// TIA Portal V17 program export: 24 tag tables, 3 data types, 17 data blocks, 29 code blocks (in call order from the OBs), 32 instance data blocks

VAR_GLOBAL   // PLC tag table "Default tag table"
   OutputPin2 AT %QB147 : Byte;
   Tag_2 AT %QB152 : Byte;
   Tag_3 AT %QB155 : Byte;
   Tag_4 AT %QB154 : Byte;
   Tag_5 AT %QB153 : Byte;
   System_Byte AT %MB0 : Byte;
   DiagStatusUpdate AT %M0.1 : Bool;
   Tag_6 AT %MW122 : UInt;
END_VAR

VAR_GLOBAL   // PLC tag table "DCmotorControlMemory"
   motorBackwardMotion AT %M1551.2 : Bool;
   motorForwardMotion AT %M1550.7 : Bool;
   motorOpposite AT %M1551.4 : Bool;
   motorMovementActive AT %M1550.6 : Bool;
   hmiTestLeftMotorAlignment AT %M1551.6 : Bool;
   hmiTestRightTrackAlignment AT %M1551.7 : Bool;
   motorDirection AT %M1550.4 : Bool;
   highPulseDone AT %M1550.5 : Bool;
   reset AT %M1552.0 : Bool;
   direction1Pulse AT %MW1500 : Int;
   ctuReset1 AT %M1550.3 : Bool;
   motorPulseWidthSelector AT %M1551.5 : Bool;
   motorPulseWIidth AT %MD1534 : DInt;
   motorCycleTime AT %MD1530 : DInt;
   motorPulseQuantity AT %MW1502 : Int;
   activateMotorOperation AT %M1550.0 : Bool;
   hmiMoveMotorForward AT %M1552.1 : Bool;
   hmiMoveMotorBackward AT %M1552.2 : Bool;
   moveMotorForward AT %M1550.1 : Bool;
   moveMotorBackward AT %M1550.2 : Bool;
   leftTrackAlignmentComplete AT %M1551.1 : Bool;
   rightTrackAlignmentComplete AT %M1551.0 : Bool;
END_VAR

VAR_GLOBAL   // PLC tag table "EKSMemory"
   userIsLogged AT %M2150.0 : Bool;
   eksUserLevel AT %MB2101 : SInt;
   ActualAuthorizationLevel AT %MB2100 : SInt;
END_VAR

VAR_GLOBAL   // PLC tag table "HMIMemory"
   currentModel AT %MW3000 : Int;
   hmiButtonVisualization AT %M3050.6 : Bool;
   previousModel AT %MW3008 : Int;
   currentStep AT %MW3002 : Int;
   numberOfStepsToMove AT %MW3006 : UInt;
   stepToDivide AT %MW3012 : UInt;
   stepToInsert AT %MW3014 : UInt;
   hmiScreenNumber AT %MW3004 : Int;
   allowedTextChange AT %M3050.0 : Bool;
   progressBarMultiply AT %MW3010 : Int;
   lastCycleInputs AT %MD3034 : DInt;
   energySavingElapsedTime AT %MD3030 : Time;
   f7Button AT %M3050.5 : Bool;
   sequencerCopySequence AT %M3050.7 : Bool;
   codeReaderConfigurationVisible AT %M3050.2 : Bool;
   analogConfigurationVisible AT %M3050.1 : Bool;
   directAlarm AT %M3050.3 : Bool;
   directHome AT %M3050.4 : Bool;
   hmiRetractClampsReady AT %M3051.0 : Bool;
END_VAR

VAR_GLOBAL   // PLC tag table "alarmMemory"
   alarm0 AT %MW100 : Int;   // alarm number
   alarm1 AT %MW102 : Int;   // alarm number
   alarm2 AT %MW104 : Int;
   retIolink AT %MW108 : Int;
   retManifold AT %MW112 : Int;
   retEuchner AT %MW106 : Int;
   retIolink2 AT %MW110 : Int;
   QuitarErrorEscaner AT %MW6 : Word;
   bypass4 AT %M2.3 : Bool;
   bypass5 AT %M2.4 : Bool;
   retPrinter AT %MW114 : Int;
   reProfinetIO1 AT %MW116 : Int;
   reProfinetIO2 AT %MW118 : Int;
   reProfinetIO3 AT %MW120 : Int;
END_VAR

VAR_GLOBAL   // PLC tag table "analogAnalysisMemory"
   leftDistanceOk AT %M1700.4 : Bool;
   rightDistanceOk AT %M1700.5 : Bool;
   leftDistanceOk2 AT %M1700.7 : Bool;
   rightDistanceOk2 AT %M1701.0 : Bool;
   initialAlignmentOK AT %M1700.1 : Bool;
   initialPositionLeftTrackOK AT %M1700.2 : Bool;
   initialPositionRightTrackOK AT %M1700.3 : Bool;
   rightDistanceNormalizedValue AT %MD1660 : Real;
   leftDistanceNormalizedValue AT %MD1664 : Real;
   leftDistanceScaledValue AT %MD1668 : Real;
   rightDistanceScaledValue AT %MD1672 : Real;
   leftEffortOk AT %M1700.0 : Bool;
   rightEffortOk AT %M1700.6 : Bool;
   leftLoadCellSensorValue AT %MW1600 : Int;
   rightLoadCellSensorValue AT %MW1602 : Int;
   leftLoadCellNormalizedValue AT %MD1676 : Real;
   rightLoadCellNormalizedValue AT %MD1680 : Real;
   leftLoadCellScaledValue AT %MD1684 : Real;
   rightLoadCellScaledValue AT %MD1688 : Real;
   leftEffortNok AT %M1701.1 : Bool;
   rightEffortNok AT %M1701.2 : Bool;
   leftTrackRemoveMessage AT %M1701.3 : Bool;
   rightTrackRemoveMessage AT %M1701.4 : Bool;
   leftLoadCellHMIStatus AT %MW1604 : Int;
   rightLoadCellHMIStatus AT %MW1606 : Int;
   leftLoadCellHMIValue AT %MD1692 : Real;
   rightLoadCellHMIValue AT %MD1696 : Real;
END_VAR

VAR_GLOBAL   // PLC tag table "clockMemory"
   Clocks200ms_FP AT %M1.1 : Bool;
   Clocks400ms_FP AT %M1.2 : Bool;
   Clocks500ms_FP AT %M1.3 : Bool;
   Clocks800ms_FP AT %M1.4 : Bool;
   Clocks1s_FP AT %M1.5 : Bool;
   Clocks1600ms_FP AT %M1.6 : Bool;
   Clocks2s_FP AT %M1.7 : Bool;
   Clocks100ms_FP AT %M1.0 : Bool;
END_VAR

VAR_GLOBAL   // PLC tag table "codeReaderMemory"
   reqScannerConfig AT %M2250.2 : Bool;
   bufferReset AT %M2250.0 : Bool;
   idleTime AT %M2250.1 : Bool;
   rightTrackLabelIdentified AT %M2250.5 : Bool;
   leftTrackLabelIdentified AT %M2250.3 : Bool;
   motorLabelIdentified AT %M2250.4 : Bool;
   labelNOK AT %M2250.6 : Bool;
   labelOK AT %M2250.7 : Bool;
   trackLabelReadOutOfNest AT %M2251.0 : Bool;
   plasticBridgeLabelReadOutOfNest AT %M2251.1 : Bool;
END_VAR

VAR_GLOBAL   // PLC tag table "modeMemory"
   automaticMode AT %M3.0 : Bool;   // AUTO = 1
   manualMode AT %M3.1 : Bool;
   noMode AT %M3.2 : Bool;
   modelChangePermit AT %M187.1 : Bool;
END_VAR

VAR_GLOBAL   // PLC tag table "permissionMemory"
   maintenacePermission AT %M4.4 : Bool;
   adminPermission AT %M4.0 : Bool;
   lgPermission AT %M4.3 : Bool;
   gapLeaderPermission AT %M4.2 : Bool;
   editingPermission AT %M4.1 : Bool;
END_VAR

VAR_GLOBAL   // PLC tag table "printerMemory"
   reqPrint AT %M4000.0 : Bool;
   reqLastLabel AT %M4000.1 : Bool;
   resetPrinterErrors AT %M4000.2 : Bool;
   printBlackLabel AT %M4000.3 : Bool;
   resetPrinterCounter AT %M4000.4 : Bool;
   hmiSavePrinterReference AT %M4000.5 : Bool;
   hmiReadPrinterReference AT %M4000.6 : Bool;
END_VAR

VAR_GLOBAL   // PLC tag table "productionMemory"
   shift1Production AT %MW300 : Int;
   shift1 AT %M350.0 : Bool;
   shift2Production AT %MW302 : Int;
   shift2 AT %M350.1 : Bool;
   shift3Production AT %MW304 : Int;
   shift3 AT %M350.2 : Bool;
   timeShift1 AT %M350.3 : Bool;
   timeShift2 AT %M350.4 : Bool;
   timeShift3 AT %M350.5 : Bool;
END_VAR

VAR_GLOBAL   // PLC tag table "programMemory"
   cycleTimeReset AT %M250.1 : Bool;
   clearData AT %M250.0 : Bool;
   programAutoModeSelection AT %M250.3 : Bool;
   productInNest AT %M250.2 : Bool;
   bypass1 AT %M2.0 : Bool;
   bypass2 AT %M2.1 : Bool;
   bypass3 AT %M2.2 : Bool;
END_VAR

VAR_GLOBAL   // PLC tag table "pulses"
   hmiPulseInt AT %MD2000 : DInt;
   HMICycleCounterRestartPulse AT %M2004.4 : Bool;
   mode01SelectedPulse AT %M2004.6 : Bool;
   model02SelectedPulse AT %M2004.7 : Bool;
   model03SelectedPulse AT %M2005.0 : Bool;
   model04SelectedPulse AT %M2005.1 : Bool;
   model05SelectedPulse AT %M2005.2 : Bool;
   model06SelectedPulse AT %M2005.3 : Bool;
   model07SelectedPulse AT %M2005.4 : Bool;
   model08SelectedPulse AT %M2005.5 : Bool;
   model09SelectedPulse AT %M2005.6 : Bool;
   model10SelectedPulse AT %M2005.7 : Bool;
   model11SelectedPulse AT %M2006.0 : Bool;
   model12SelectedPulse AT %M2006.1 : Bool;
   model13SelectedPulse AT %M2006.2 : Bool;
   model14SelectedPulse AT %M2006.3 : Bool;
   model15SelectedPulse AT %M2006.4 : Bool;
   alarmPresentPulse AT %M2004.3 : Bool;
   "1stShiftChangePulse" AT %M2004.0 : Bool;
   "2ndShiftChangePulse" AT %M2004.1 : Bool;
   "3rdShiftChangePulse" AT %M2004.2 : Bool;
   stepChangeTimerResetInputPulse AT %M2009.4 : Bool;
   stepChangeTimerResetOutputPulse AT %M2009.5 : Bool;
   stationTurnedOffInSequencePulse AT %M2009.3 : Bool;
   model32SelectedPulse AT %M2008.5 : Bool;
   model31SelectedPulse AT %M2008.4 : Bool;
   model30SelectedPulse AT %M2008.3 : Bool;
   model29SelectedPulse AT %M2008.2 : Bool;
   model27SelectedPulse AT %M2008.0 : Bool;
   model28SelectedPulse AT %M2008.1 : Bool;
   model26SelectedPulse AT %M2007.7 : Bool;
   model25SelectedPulse AT %M2007.6 : Bool;
   model24SelectedPulse AT %M2007.5 : Bool;
   model23SelectedPulse AT %M2007.4 : Bool;
   model22SelectedPulse AT %M2007.3 : Bool;
   model21SelectedPulse AT %M2007.2 : Bool;
   model20SelectedPulse AT %M2007.1 : Bool;
   model19SelectedPulse AT %M2007.0 : Bool;
   model18SelectedPulse AT %M2006.7 : Bool;
   model17SelectedPulse AT %M2006.6 : Bool;
   model16SelectedPulse AT %M2006.5 : Bool;
   scanner3DataLogPulse AT %M2009.2 : Bool;
   scanner2DataLogPulse AT %M2009.1 : Bool;
   scanner1DataLogPulse AT %M2009.0 : Bool;
   motorScannerPulse AT %M2008.6 : Bool;
   rightTrackScannerPulse AT %M2008.7 : Bool;
   leftTrackScannerPulse AT %M2004.5 : Bool;
   scannerOk1Pulse AT %M2009.6 : Bool;
   scannerOk2Pulse AT %M2009.7 : Bool;
   scannerOk3Pulse AT %M2010.0 : Bool;
   leftTrackNokAlarmPulse AT %M2010.1 : Bool;
   rightTrackNokAlarmPulse AT %M2010.2 : Bool;
END_VAR

VAR_GLOBAL   // PLC tag table "sequenceMemory"
   aa AT %MW1104 : Int;
   a_correctas AT %MW1100 : Int;
   a_estados AT %MW1102 : Int;
   verificacion_estados_A AT %MW1114 : Int;
   verificacion_estados_B AT %MW1116 : Int;
   b_estados AT %MW1106 : Int;
   numberOfCorrectOutputStates AT %MW1110 : Int;
   bb AT %MW1108 : Int;
   previousStep AT %MW1112 : Int;
   sequenceRestart AT %M1150.0 : Bool;
   stationTurnedOffInSequence AT %M1150.1 : Bool;
END_VAR

VAR_GLOBAL   // PLC tag table "systemMemory"
   firstScan AT %M0.0 : Bool;
   LOG1 AT %M0.2 : Bool;
   LOG0 AT %M0.3 : Bool;
END_VAR

VAR_GLOBAL   // PLC tag table "EKSFieldbusInputs"
   iEKSLevel AT %IB201 : Byte;
   iEKSChipInside AT %I200.1 : Bool;
   iEKSEmployeeNumber AT %ID221 : DWord;
   iEKSKeyID1 AT %ID320 : DWord;
   iEKSKeyID2 AT %ID324 : DWord;
   iEKSJobFinished AT %I200.6 : Bool;
END_VAR

VAR_GLOBAL   // PLC tag table "safetyControllerFieldbusInputs"
   iSecurityEnabled AT %I46.0 : Bool;
   iEmergencyStop AT %I62.0 : Bool;
   iEmergencyStopMonitor AT %I62.1 : Bool;
   iOutputsEnabled AT %I82.0 : Bool;
END_VAR

VAR_GLOBAL   // PLC tag table "analogPLCInputs"
   iLeftLoadCell AT %IW13 : Int;
   iRightLoadCell AT %IW15 : Int;
   iRightDistanceSensor AT %IW17 : Int;
   iLeftDistanceSensor AT %IW19 : UInt;
END_VAR

VAR_GLOBAL   // PLC tag table "digitalFieldbusInputs"
   iRightTrackClampExt AT %I147.0 : Bool;
   iLeftTrackClampExt AT %I147.1 : Bool;
   iRightNestLocatingPinExt AT %I147.2 : Bool;
   iLeftNestLocatingPinExt AT %I147.3 : Bool;
   iRightTrackClampRet AT %I148.0 : Bool;
   iLeftTrackClampRet AT %I148.1 : Bool;
   iRightNestLocatingPinRet AT %I148.2 : Bool;
   iLeftNestLocatingPinRet AT %I148.3 : Bool;
   iLeftTrackPS1 AT %I149.0 : Bool;
   iLeftTrackPS2 AT %I149.1 : Bool;
   iRightTrackPS1 AT %I149.2 : Bool;
   iRightTrackPS2 AT %I149.3 : Bool;
   iLeftNestInitialPos AT %I149.4 : Bool;
   iRightNestInitialPos AT %I149.5 : Bool;
   iRightManualClampClosed AT %I149.6 : Bool;
   iLeftManualClampClosed AT %I149.7 : Bool;
   iPlasticBridgePS AT %I151.0 : Bool;
   iLeftNestWorkingPos AT %I151.1 : Bool;
   iPokayokeLeftTrackPS AT %I151.2 : Bool;
   iPokayokeRightTrackPS AT %I151.3 : Bool;
   iPlasticBridgeClampClosed AT %I151.4 : Bool;
   iInsertPlasticBridgePos AT %I151.6 : Bool;
   iInsertShaftPos AT %I151.7 : Bool;
END_VAR

VAR_GLOBAL   // PLC tag table "digitalPLCInputs"
   iAirPreassureSensor AT %I0.1 : Bool;
   iMotorConnected AT %I0.2 : Bool;
   iRestartButton AT %I0.0 : Bool;
   iMotorRelayStatus AT %I0.3 : Bool;
END_VAR

VAR_GLOBAL   // PLC tag table "digitalFielbusOutputs"
   qCylinder1DirectionA AT %Q149.0 : Bool;
   qCylinder1DirectionB AT %Q151.0 : Bool;
   qCylinder2DirectionA AT %Q149.1 : Bool;
   qCylinder2DirectionB AT %Q151.1 : Bool;
   qCylinder7DirectionA AT %Q149.6 : Bool;
   qCylinder7DirectionB AT %Q151.6 : Bool;
   qCylinder4DirectionA AT %Q149.3 : Bool;
   qCylinder4DirectionB AT %Q151.3 : Bool;
   qCylinder5DirectionA AT %Q149.4 : Bool;
   qCylinder5DirectionB AT %Q151.4 : Bool;
   qCylinder6DirectionA AT %Q149.5 : Bool;
   qCylinder6DirectionB AT %Q151.5 : Bool;
   qCylinder3DirectionA AT %Q149.2 : Bool;
   qCylinder3DirectionB AT %Q151.2 : Bool;
   qCylinder8DirectionA AT %Q149.7 : Bool;
   qCylinder8DirectionB AT %Q151.7 : Bool;
   qCylinder9DirectionA AT %Q148.0 : Bool;
   qCylinder9DirectionB AT %Q150.0 : Bool;
   qCylinder10DirectionA AT %Q148.1 : Bool;
   qCylinder10DirectionB AT %Q150.1 : Bool;
   qActivateCutOffValve AT %Q147.0 : Bool;
END_VAR

VAR_GLOBAL   // PLC tag table "digitalPLCOutputs"
   qAirInletValve AT %Q0.0 : Bool;
   qLampActivation AT %Q0.4 : Bool;
   qFanActivation AT %Q0.5 : Bool;
   qRedStacklight AT %Q1.7 : Bool;
   qYellowStacklight AT %Q1.6 : Bool;
   qGreenStacklight AT %Q1.5 : Bool;
   qControlIN AT %Q0.6 : Bool;
   qActiveMotor AT %Q0.7 : Bool;
   qDirectionChange AT %Q1.0 : Bool;
   qRedIndicator AT %Q1.1 : Bool;
   qGreenIndicator AT %Q1.2 : Bool;
   qYellowIndicator AT %Q1.3 : Bool;
   qBlueStacklight AT %Q1.4 : Bool;
END_VAR

VAR_GLOBAL   // PLC tag table "EKSFieldbusOutputs"
   qEKSStartAddress AT %QB201 : Byte;
   qEKSDataLength AT %QB202 : Byte;
   qEKSData1 AT %QB204 : Byte;
   qEKSData2 AT %QB205 : Byte;
   qEKSWriteCMD AT %Q200.0 : Bool;
END_VAR

TYPE "udtButtons"
// stored: IsFailsafeCompliant false
   STRUCT
      bReq : Bool;
      bP : Bool;
      bTGG : Bool;
      bCmd : Bool;
      bAkn : Bool;
      b1 : Bool;
      b2 : Bool;
      b3 : Bool;
   END_STRUCT;
END_TYPE

TYPE "udt_EKS_KEY"
// stored: IsFailsafeCompliant false
   STRUCT
      ID1 : DWord;   // Key unique ID [bytes 1-4]
      ID2 : DWord;   // Key unique ID [bytes 5-8]
      EMPLOYEE_ID : DWord;   // Employee ID number [hex format]
      LEVEL : Int;   // Key level stored inside key
      COMMENTS : WString[10];   // Comments of the key
      _res_1 : Int;
   END_STRUCT;
END_TYPE

TYPE "udt_referenceMainInfo"
// stored: IsFailsafeCompliant false
   STRUCT
      id : Int;
      description : String[20];
      partNumber : String[8];
      rev : String[2];
      customerNumber : String[8];
      vpps : String[14];
      locationCode : String[1];
      dataIdentifier : String[3];
      duns : String[9];
   END_STRUCT;
END_TYPE

DATA_BLOCK "DB_REC_IJCORE"   // DB1006
{ S7_Optimized_Access := 'FALSE' }
VERSION : 0.1
// stored: AutoNumber false, DBAccessibleFromOPCUA true, DBAccessibleFromWebserver true, IsOnlyStoredInLoadMemory false, IsWriteProtectedInAS false
   VAR
      SW_Message : Array[1..300] of Word;
      Message : Array[1..50] of Struct
         Answer : Int;
         Content : Array[1..30] of Byte;
      END_STRUCT;
   END_VAR
BEGIN
   SW_Message[1..8] := 16#FFFF;
   SW_Message[9..300] := 16#0000;
   Message[1..50].Answer := 0;
   Message[1].Content[1..30] := 16#00;
   Message[2].Content[1..30] := 16#00;
   Message[3].Content[1..30] := 16#00;
   Message[4].Content[1..30] := 16#00;
   Message[5].Content[1..30] := 16#00;
   Message[6].Content[1..30] := 16#00;
   Message[7].Content[1..30] := 16#00;
   Message[8].Content[1..30] := 16#00;
   Message[9].Content[1..30] := 16#00;
   Message[10].Content[1..30] := 16#00;
   Message[11].Content[1..30] := 16#00;
   Message[12].Content[1..30] := 16#00;
   Message[13].Content[1..30] := 16#00;
   Message[14].Content[1..30] := 16#00;
   Message[15].Content[1..30] := 16#00;
   Message[16].Content[1..30] := 16#00;
   Message[17].Content[1..30] := 16#00;
   Message[18].Content[1..30] := 16#00;
   Message[19].Content[1..30] := 16#00;
   Message[20].Content[1..30] := 16#00;
   Message[21].Content[1..30] := 16#00;
   Message[22].Content[1..30] := 16#00;
   Message[23].Content[1..30] := 16#00;
   Message[24].Content[1..30] := 16#00;
   Message[25].Content[1..30] := 16#00;
   Message[26].Content[1..30] := 16#00;
   Message[27].Content[1..30] := 16#00;
   Message[28].Content[1..30] := 16#00;
   Message[29].Content[1..30] := 16#00;
   Message[30].Content[1..30] := 16#00;
   Message[31].Content[1..30] := 16#00;
   Message[32].Content[1..30] := 16#00;
   Message[33].Content[1..30] := 16#00;
   Message[34].Content[1..30] := 16#00;
   Message[35].Content[1..30] := 16#00;
   Message[36].Content[1..30] := 16#00;
   Message[37].Content[1..30] := 16#00;
   Message[38].Content[1..30] := 16#00;
   Message[39].Content[1..30] := 16#00;
   Message[40].Content[1..30] := 16#00;
   Message[41].Content[1..30] := 16#00;
   Message[42].Content[1..30] := 16#00;
   Message[43].Content[1..30] := 16#00;
   Message[44].Content[1..30] := 16#00;
   Message[45].Content[1..30] := 16#00;
   Message[46].Content[1..30] := 16#00;
   Message[47].Content[1..30] := 16#00;
   Message[48].Content[1..30] := 16#00;
   Message[49].Content[1..30] := 16#00;
   Message[50].Content[1..30] := 16#00;
END_DATA_BLOCK

DATA_BLOCK "DB_SEND_IJCORE"   // DB1005
{ S7_Optimized_Access := 'FALSE' }
VERSION : 0.1
// stored: AutoNumber false, DBAccessibleFromOPCUA true, DBAccessibleFromWebserver true, IsOnlyStoredInLoadMemory false, IsWriteProtectedInAS false
   VAR
      Awake_DW : Word := 16#0000;
      Awake_SW : Int := 1;
      SW_Message : Array[1..300] of Word;
      Message : Array[1..50] of Struct
         Content : Array[1..80] of Byte;
      END_STRUCT;
   END_VAR
BEGIN
   SW_Message[1..8] := 16#FFFF;
   SW_Message[9..300] := 16#0000;
   Message[1].Content[1..80] := 16#00;
   Message[2].Content[1..80] := 16#00;
   Message[3].Content[1..80] := 16#00;
   Message[4].Content[1..80] := 16#00;
   Message[5].Content[1..80] := 16#00;
   Message[6].Content[1..80] := 16#00;
   Message[7].Content[1..80] := 16#00;
   Message[8].Content[1..80] := 16#00;
   Message[9].Content[1..80] := 16#00;
   Message[10].Content[1..80] := 16#00;
   Message[11].Content[1..80] := 16#00;
   Message[12].Content[1..80] := 16#00;
   Message[13].Content[1..80] := 16#00;
   Message[14].Content[1..80] := 16#00;
   Message[15].Content[1..80] := 16#00;
   Message[16].Content[1..80] := 16#00;
   Message[17].Content[1..80] := 16#00;
   Message[18].Content[1..80] := 16#00;
   Message[19].Content[1..80] := 16#00;
   Message[20].Content[1..80] := 16#00;
   Message[21].Content[1..80] := 16#00;
   Message[22].Content[1..80] := 16#00;
   Message[23].Content[1..80] := 16#00;
   Message[24].Content[1..80] := 16#00;
   Message[25].Content[1..80] := 16#00;
   Message[26].Content[1..80] := 16#00;
   Message[27].Content[1..80] := 16#00;
   Message[28].Content[1..80] := 16#00;
   Message[29].Content[1..80] := 16#00;
   Message[30].Content[1..80] := 16#00;
   Message[31].Content[1..80] := 16#00;
   Message[32].Content[1..80] := 16#00;
   Message[33].Content[1..80] := 16#00;
   Message[34].Content[1..80] := 16#00;
   Message[35].Content[1..80] := 16#00;
   Message[36].Content[1..80] := 16#00;
   Message[37].Content[1..80] := 16#00;
   Message[38].Content[1..80] := 16#00;
   Message[39].Content[1..80] := 16#00;
   Message[40].Content[1..80] := 16#00;
   Message[41].Content[1..80] := 16#00;
   Message[42].Content[1..80] := 16#00;
   Message[43].Content[1..80] := 16#00;
   Message[44].Content[1..80] := 16#00;
   Message[45].Content[1..80] := 16#00;
   Message[46].Content[1..80] := 16#00;
   Message[47].Content[1..80] := 16#00;
   Message[48].Content[1..80] := 16#00;
   Message[49].Content[1..80] := 16#00;
   Message[50].Content[1..80] := 16#00;
END_DATA_BLOCK

DATA_BLOCK "model"   // DB5
{ S7_Optimized_Access := 'TRUE' }
VERSION : 0.1
// stored: AutoNumber false, DBAccessibleFromOPCUA true, DBAccessibleFromWebserver true, IsOnlyStoredInLoadMemory false, IsRetainMemResEnabled false, IsWriteProtectedInAS false, MemoryReserve 100
   VAR RETAIN
      "name" : Array[0..32] of String[50];
   END_VAR
   VAR
      day : Int := 2;
      dayText : String := '    11';
      month : Int := 8;
      monthText : String := '     8';
      year : Int := 2012;
      yearReady : String := '2012';
      hour : Int := 17;
      hourText : String := '    17';
      minutes : Int := 30;
      minutesText : String := '    30';
      seconds : Int := 30;
      secondsText : String := '    31';
      active : Array[0..32] of Bool;
   END_VAR
   VAR RETAIN
      datum1 : Array[0..32] of String[50];
      datum2 : Array[0..32] of String[50];
      datum3 : Array[0..32] of String[50];
      datum4 : Array[0..32] of String[50];
      datum5 : Array[0..32] of String[50];
      datum6 : Array[0..32] of String[50];
      datum7 : Array[0..32] of String[50];
      Description : Array[0..32] of String[50];
   END_VAR
BEGIN
   "name"[0..1] := '4118099';
   "name"[2] := '4118098';
   "name"[3..32] := '';
   active[0] := FALSE;
   active[1..2] := TRUE;
   active[3..32] := FALSE;
   datum1[0..2] := 'Z';
   datum1[3] := 'ddd';
   datum1[4..17] := 'Z';
   datum1[18..32] := '';
   datum2[0..17] := '410';
   datum2[18..32] := '';
   datum3[0..17] := '6';
   datum3[18..32] := '';
   datum4[0..2] := 'BACKREST W33A POWER MEMO L6';
   datum4[3] := 'prueba';
   datum4[4] := 'outter trackw33';
   datum4[5..16] := 'BACKREST W33A POWER MEMO L6';
   datum4[17] := 'P42LHNOMEM';
   datum4[18..32] := '';
   datum5[0] := '2389161X-01';
   datum5[1..2] := '2521784';
   datum5[3] := '2389161X-01';
   datum5[4..5] := '2282685X-01';
   datum5[6..16] := '2521784';
   datum5[17] := '2418723X-01';
   datum5[18..32] := '';
   datum6[0..32] := '';
   datum7[0..32] := '';
   Description[0..1] := 'H-Frame 4W RH';
   Description[2] := 'H-Frame 4W LH';
   Description[3..32] := '';
END_DATA_BLOCK

DATA_BLOCK "retentiveValues"   // DB54
{ S7_Optimized_Access := 'TRUE' }
VERSION : 0.1
// stored: AutoNumber true, DBAccessibleFromOPCUA true, DBAccessibleFromWebserver true, IsOnlyStoredInLoadMemory false, IsRetainMemResEnabled true, IsWriteProtectedInAS false, MemoryReserve 100, RetainMemoryReserve 0
   VAR RETAIN
      stationInSequence : Bool := FALSE;
   END_VAR
BEGIN
END_DATA_BLOCK

DATA_BLOCK "analog"   // DB3
{ S7_Optimized_Access := 'TRUE' }
VERSION : 0.1
// stored: AutoNumber false, DBAccessibleFromOPCUA true, DBAccessibleFromWebserver true, IsOnlyStoredInLoadMemory false, IsRetainMemResEnabled false, IsWriteProtectedInAS false, MemoryReserve 100
   VAR RETAIN
      value1 : Array[0..32] of Real;   // Setpoint del valor analógico 1 [modelo]
      low1 : Array[0..32] of Real;   // Valor bajo del valor analógico 1 [modelo]
      high1 : Array[0..32] of Real;   // Valor alto del valor analógico 1 [modelo]
      value2 : Array[0..32] of Real;
      low2 : Array[0..32] of Real;
      high2 : Array[0..32] of Real;
      value3 : Array[0..32] of Real;
      low3 : Array[0..32] of Real;
      high3 : Array[0..32] of Real;
      value4 : Array[0..32] of Real;
      low4 : Array[0..32] of Real;
      high4 : Array[0..32] of Real;
      value5 : Array[0..32] of Real;
      low5 : Array[0..32] of Real;
      high5 : Array[0..32] of Real;
      value6 : Array[0..32] of Real;
      low6 : Array[0..32] of Real;
      high6 : Array[0..32] of Real;
      value7 : Array[0..32] of Real;
      low7 : Array[0..32] of Real;
      high7 : Array[0..32] of Real;
      value8 : Array[0..32] of Real;
      low8 : Array[0..32] of Real;
      high8 : Array[0..32] of Real;
      value9 : Array[0..32] of Real;
      low9 : Array[0..32] of Real;
      high9 : Array[0..32] of Real;
      value10 : Array[0..32] of Real;
      low10 : Array[0..32] of Real;
      high10 : Array[0..32] of Real;
      text : Array[0..10] of String;
      analog1 : Bool := TRUE;
      analog2 : Bool := TRUE;
      analog3 : Bool := TRUE;
      analog4 : Bool := TRUE;
      analog5 : Bool := FALSE;
      analog6 : Bool := FALSE;
   END_VAR
   VAR
      visibility : Array[0..6] of Bool;
      current1 : Int := 0;
      current2 : Int := 0;
      current3 : Int := 0;
      current4 : Int := 0;
      current5 : Int := 0;
      current6 : Int := 0;
      laserConstant : Real := 0.005802801;
      okDistance : Bool := FALSE;
      nest1 : Array[0..5] of Int;
      nest2 : Array[0..5] of Int;
      nest3 : Array[0..5] of Int;
      nest4 : Array[0..5] of Int;
      motorCounter : Int := 1600;
   END_VAR
   VAR RETAIN
      motorQuantity : Int := 0;
   END_VAR
   VAR
      analogReading1 : Array[0..9] of Real;
      analogReading2 : Array[0..9] of Real;
      leftLoadCellMaxValueObtained : Real := 0.0;
      rightLoadCellMaxValueObtained : Real := 0.0;
   END_VAR
BEGIN
   value1[0..3] := -63.9458;
   value1[4] := -16.86112;
   value1[5..8] := -63.9458;
   value1[9..14] := 131.4746;
   value1[15] := 340.0;
   value1[16] := -17.19834;
   value1[17..19] := 131.4746;
   value1[20..32] := 0.0;
   low1[0..2] := -1.0;
   low1[3] := 120.0;
   low1[4] := 154.0;
   low1[5] := 100.0;
   low1[6..8] := 72.0;
   low1[9..13] := 120.0;
   low1[14] := 153.0;
   low1[15] := 0.0;
   low1[16..17] := 120.0;
   low1[18] := 154.0;
   low1[19] := 120.0;
   low1[20..32] := 0.0;
   high1[0..2] := 2.0;
   high1[3] := 5.0;
   high1[4] := 2.0;
   high1[5] := 110.0;
   high1[6..8] := 76.0;
   high1[9..13] := 5.0;
   high1[14] := 2.0;
   high1[15] := 41.1;
   high1[16..17] := 5.0;
   high1[18] := 2.0;
   high1[19] := 5.0;
   high1[20..32] := 0.0;
   value2[0..3] := -65.29469;
   value2[4] := -17.51449;
   value2[5..8] := -65.29469;
   value2[9..14] := 131.4746;
   value2[15] := 340.0;
   value2[16] := -17.40911;
   value2[17..19] := 131.4746;
   value2[20..32] := 0.0;
   low2[0..2] := -1.0;
   low2[3] := 60.0;
   low2[4] := 154.0;
   low2[5] := 100.0;
   low2[6..8] := 60.0;
   low2[9..13] := 0.0;
   low2[14] := 153.0;
   low2[15..17] := 0.0;
   low2[18] := 154.0;
   low2[19..32] := 0.0;
   high2[0..2] := 2.0;
   high2[3] := 75.0;
   high2[4] := 2.0;
   high2[5] := 110.0;
   high2[6..8] := 64.0;
   high2[9..13] := 5.0;
   high2[14] := 2.0;
   high2[15] := 38.7;
   high2[16..17] := 5.0;
   high2[18] := 2.0;
   high2[19] := 5.0;
   high2[20..32] := 0.0;
   value3[0..3] := 16#0000_02E7;
   value3[4] := 16#0000_01DE;
   value3[5..8] := 16#0000_02E7;
   value3[9..14] := 16#0000_01DE;
   value3[15..16] := 16#0000_DDDE;
   value3[17..19] := 16#0000_01DE;
   value3[20..32] := 0.0;
   low3[0..2] := 200.0;
   low3[3] := 40.0;
   low3[4] := 0.0;
   low3[5] := 200.0;
   low3[6..8] := 40.0;
   low3[9..32] := 0.0;
   high3[0..2] := 500.0;
   high3[3] := 250.0;
   high3[4] := 0.0;
   high3[5] := 210.0;
   high3[6..8] := 250.0;
   high3[9..32] := 0.0;
   value4[0..19] := 40.0;
   value4[20..32] := 0.0;
   low4[0..2] := 200.0;
   low4[3] := 40.0;
   low4[4] := 0.0;
   low4[5] := 200.0;
   low4[6..8] := 40.0;
   low4[9..32] := 0.0;
   high4[0..2] := 500.0;
   high4[3] := 250.0;
   high4[4] := 3.0;
   high4[5] := 210.0;
   high4[6..8] := 250.0;
   high4[9..19] := 3.0;
   high4[20..32] := 0.0;
   value5[0..14] := 3.0;
   value5[15] := 8.0;
   value5[16..19] := 3.0;
   value5[20..32] := 0.0;
   low5[0..32] := 0.0;
   high5[0..19] := 59.0;
   high5[20..32] := 0.0;
   value6[0..32] := 0.0;
   low6[0..32] := 0.0;
   high6[0..32] := 0.0;
   value7[0..3] := -65.29469;
   value7[4] := -16.90327;
   value7[5..8] := -65.29469;
   value7[9..14] := -16.86112;
   value7[15] := 0.0;
   value7[16] := -17.19834;
   value7[17..19] := -16.86112;
   value7[20..32] := 0.0;
   low7[0..3] := 142.0;
   low7[4] := 125.0;
   low7[5..8] := 142.0;
   low7[9..13] := 0.0;
   low7[14] := 26.0;
   low7[15..17] := 0.0;
   low7[18] := 128.0;
   low7[19..32] := 0.0;
   high7[0..3] := 2.0;
   high7[4] := 3.0;
   high7[5..13] := 2.0;
   high7[14] := 5.0;
   high7[15] := 0.0;
   high7[16..19] := 2.0;
   high7[20..32] := 0.0;
   value8[0..3] := -65.29469;
   value8[4] := -17.17727;
   value8[5..8] := -65.29469;
   value8[9..14] := -17.17727;
   value8[15] := 0.0;
   value8[16] := -17.51449;
   value8[17..19] := -17.17727;
   value8[20..32] := 0.0;
   low8[0..3] := 142.0;
   low8[4] := 125.0;
   low8[5..8] := 142.0;
   low8[9..13] := 0.0;
   low8[14] := 26.0;
   low8[15..17] := 0.0;
   low8[18] := 128.0;
   low8[19..32] := 0.0;
   high8[0..3] := 2.0;
   high8[4] := 3.0;
   high8[5..13] := 2.0;
   high8[14] := 5.0;
   high8[15] := 0.0;
   high8[16..19] := 2.0;
   high8[20..32] := 0.0;
   value9[0..3] := 1.348892;
   value9[4] := 0.6533699;
   value9[5..8] := 1.348892;
   value9[9..32] := 0.0;
   low9[0..32] := 0.0;
   high9[0..3] := 0.0;
   high9[4] := 2.0;
   high9[5..13] := 0.0;
   high9[14] := 2.0;
   high9[15..17] := 0.0;
   high9[18] := 2.0;
   high9[19..32] := 0.0;
   value10[0..3] := 0.0;
   value10[4] := 0.2739925;
   value10[5..8] := 0.0;
   value10[9..14] := 0.3161469;
   value10[15..16] := 0.0;
   value10[17..19] := 0.3161469;
   value10[20..32] := 0.0;
   low10[0..32] := 0.0;
   high10[0..17] := 0.0;
   high10[18] := 2.0;
   high10[19..32] := 0.0;
   text[0] := '';
   text[1] := 'Distancia Izquierda';
   text[2] := 'Distancia Derecha';
   text[3] := 'Esfuerzo Izquierdo';
   text[4] := 'Esfuerzo Derecho';
   text[5..6] := '';
   text[7] := 'Final izquierdo';
   text[8] := 'Final derecho';
   text[9] := 'Alineacion inicial';
   text[10] := 'Alineacion final';
   visibility[0] := FALSE;
   visibility[1..4] := TRUE;
   visibility[5..6] := FALSE;
   nest1[0..5] := 0;
   nest2[0..5] := 0;
   nest3[0..5] := 0;
   nest4[0..5] := 0;
   analogReading1[0..2] := 58.96373;
   analogReading1[3] := 0.4987493;
   analogReading1[4] := 0.0;
   analogReading1[5..9] := 58.96373;
   analogReading2[0..9] := 0.0;
END_DATA_BLOCK

DATA_BLOCK "eks"   // DB305
{ S7_Optimized_Access := 'FALSE' }
VERSION : 0.1
// stored: AutoNumber false, DBAccessibleFromOPCUA true, DBAccessibleFromWebserver true, IsOnlyStoredInLoadMemory false, IsWriteProtectedInAS false
   VAR RETAIN
      status : Struct
         operator : Bool := TRUE;
         gapLeader : Bool := TRUE;
         maintenance : Bool := TRUE;
         administrator : Bool := TRUE;
         spare4 : Bool := FALSE;
         spare5 : Bool := FALSE;
         spare6 : Bool := FALSE;
         spare7 : Bool := FALSE;
         addModeEnabled : Bool := TRUE;
         addMode : Bool := FALSE;
         reset : Bool := FALSE;
         nbMaxAchieved : Bool := FALSE;
         fpStoreKeyIn : Bool := FALSE;
         spare15 : Bool := FALSE;
         spare16 : Bool := FALSE;
         spare17 : Bool := FALSE;
      END_STRUCT;
      hmi : Struct
         operatorKey : Bool := FALSE;
         addMode : Bool := FALSE;
         endAddMode : Bool := FALSE;
         writeKeyNewLevel : Bool := FALSE;
         writeKewKeyID : Bool := FALSE;
         updateNbAdmin : Bool := FALSE;
         spare6 : Bool := FALSE;
         spare7 : Bool := FALSE;
         spare10 : Bool := FALSE;
         spare11 : Bool := FALSE;
         spare12 : Bool := FALSE;
         spare13 : Bool := FALSE;
         spare14 : Bool := FALSE;
         spare15 : Bool := FALSE;
         spare16 : Bool := FALSE;
         spare17 : Bool := FALSE;
      END_STRUCT;
      timeout : Struct
         resetSet : Int := 9999;
         resetStatus : Int := 9100;
      END_STRUCT;
      pageIndex : Int := 1;   // Index of the page of HMI
      saveLine : Int := 0;   // Line to save key
      removeLine : Int := 0;   // Line to remove key
      actualLevel : Int := 5;   // Actual level of key
      nbAdmin : Int := 30740;   // Number of admin counted
      tCycle : Int := 0;   // Index for function Cycle (look for key)
      nbMaxAdmin : Int := 5;   // Number of administrator max
      savedPageNumber : Word := 16#0001;
      sparesBlock1 : Array[22..47] of Byte;   // Reserve
      insertedKey { S7_SetPoint := 'True'} : "udt_EKS_KEY";   // Information of Key Inserted
      hmiPage { S7_SetPoint := 'True'} : Array[1..10] of "udt_EKS_KEY";   // Information displayed on HMI
      spareBlock2 : Array[270..299] of Byte;   // Reserve
      keys { S7_SetPoint := 'True'} : Array[1..130] of "udt_EKS_KEY";
      deleteKeys : "udt_EKS_KEY";
   END_VAR
BEGIN
   sparesBlock1[22..47] := 16#00;
   insertedKey.ID1 := 16#6B8F_0010;
   insertedKey.ID2 := 16#3200_0000;
   insertedKey.EMPLOYEE_ID := 16#0000_0000;
   insertedKey.LEVEL := 5;
   insertedKey.COMMENTS := WSTRING#'ADMIN';
   insertedKey._res_1 := 0;
   hmiPage[1].ID1 := 16#27A0_0010;
   hmiPage[2].ID1 := 16#8DDD_0010;
   hmiPage[3].ID1 := 16#9750_0010;
   hmiPage[4].ID1 := 16#4D33_0010;
   hmiPage[5].ID1 := 16#7650_0010;
   hmiPage[6].ID1 := 16#6B8F_0010;
   hmiPage[7].ID1 := 16#3A6D_0010;
   hmiPage[8..10].ID1 := 16#0000_0000;
   hmiPage[1..7].ID2 := 16#3200_0000;
   hmiPage[8..10].ID2 := 16#0000_0000;
   hmiPage[1].EMPLOYEE_ID := 16#0001_0000;
   hmiPage[2].EMPLOYEE_ID := 16#0000_0001;
   hmiPage[3].EMPLOYEE_ID := 16#0000_0002;
   hmiPage[4..5].EMPLOYEE_ID := 16#0000_0000;
   hmiPage[6].EMPLOYEE_ID := 16#0000_0200;
   hmiPage[7].EMPLOYEE_ID := 16#0000_0100;
   hmiPage[8..10].EMPLOYEE_ID := 16#0000_0000;
   hmiPage[1].LEVEL := 5;
   hmiPage[2].LEVEL := 2;
   hmiPage[3].LEVEL := 3;
   hmiPage[4].LEVEL := 5;
   hmiPage[5].LEVEL := 3;
   hmiPage[6].LEVEL := 5;
   hmiPage[7].LEVEL := 3;
   hmiPage[8..10].LEVEL := 0;
   hmiPage[1].COMMENTS := WSTRING#'CESAR';
   hmiPage[2].COMMENTS := WSTRING#'GAP';
   hmiPage[3].COMMENTS := WSTRING#'MANT';
   hmiPage[4..5].COMMENTS := WSTRING#'CESAR';
   hmiPage[6].COMMENTS := WSTRING#'ADMIN';
   hmiPage[7].COMMENTS := WSTRING#'MANT';
   hmiPage[8..10].COMMENTS := WSTRING#'';
   hmiPage[1..10]._res_1 := 0;
   spareBlock2[270..299] := 16#00;
   keys[1].ID1 := 16#27A0_0010;
   keys[2].ID1 := 16#8DDD_0010;
   keys[3].ID1 := 16#9750_0010;
   keys[4].ID1 := 16#4D33_0010;
   keys[5].ID1 := 16#7650_0010;
   keys[6].ID1 := 16#6B8F_0010;
   keys[7].ID1 := 16#3A6D_0010;
   keys[8..109].ID1 := 16#0000_0000;
   keys[110].ID1 := 16#DB52_0010;
   keys[111..130].ID1 := 16#0000_0000;
   keys[1..7].ID2 := 16#3200_0000;
   keys[8..109].ID2 := 16#0000_0000;
   keys[110].ID2 := 16#3200_0000;
   keys[111..130].ID2 := 16#0000_0000;
   keys[1].EMPLOYEE_ID := 16#0001_0000;
   keys[2].EMPLOYEE_ID := 16#0000_0001;
   keys[3].EMPLOYEE_ID := 16#0000_0002;
   keys[4..5].EMPLOYEE_ID := 16#0000_0000;
   keys[6].EMPLOYEE_ID := 16#0000_0200;
   keys[7].EMPLOYEE_ID := 16#0000_0100;
   keys[8..130].EMPLOYEE_ID := 16#0000_0000;
   keys[1].LEVEL := 5;
   keys[2].LEVEL := 2;
   keys[3].LEVEL := 3;
   keys[4].LEVEL := 5;
   keys[5].LEVEL := 3;
   keys[6].LEVEL := 5;
   keys[7].LEVEL := 3;
   keys[8..109].LEVEL := 0;
   keys[110].LEVEL := 5;
   keys[111..130].LEVEL := 0;
   keys[1].COMMENTS := WSTRING#'CESAR';
   keys[2].COMMENTS := WSTRING#'GAP';
   keys[3].COMMENTS := WSTRING#'MANT';
   keys[4..5].COMMENTS := WSTRING#'CESAR';
   keys[6].COMMENTS := WSTRING#'ADMIN';
   keys[7].COMMENTS := WSTRING#'MANT';
   keys[8..109].COMMENTS := WSTRING#'';
   keys[110].COMMENTS := WSTRING#'Robins';
   keys[111..130].COMMENTS := WSTRING#'';
   keys[1..130]._res_1 := 0;
   deleteKeys.ID1 := 16#0000_0000;
   deleteKeys.ID2 := 16#0000_0000;
   deleteKeys.EMPLOYEE_ID := 16#0000_0000;
   deleteKeys.LEVEL := 0;
   deleteKeys.COMMENTS := WSTRING#'';
   deleteKeys._res_1 := 0;
END_DATA_BLOCK

DATA_BLOCK "motor"   // DB19
{ S7_Optimized_Access := 'TRUE' }
VERSION : 0.1
// stored: AutoNumber true, DBAccessibleFromOPCUA true, DBAccessibleFromWebserver true, IsOnlyStoredInLoadMemory false, IsRetainMemResEnabled false, IsWriteProtectedInAS false, MemoryReserve 100
   VAR RETAIN
      on : Bool := TRUE;
      track1Test : Bool := FALSE;
      track2Test : Bool := FALSE;
      pulseNumber1 : Int := 5;
      waitTime1 : DInt := 100;
      pulseWidth2 : DInt := 10;
      cicleTime2 : DInt := 200;
      pulseNumber2 : Int := 5;
      waitTime2 : DInt := 100;
      cicleTime1 : DInt := 200;
      pulseWidth1 : DInt := 10;
   END_VAR
BEGIN
END_DATA_BLOCK

DATA_BLOCK "step"   // DB4
{ S7_Optimized_Access := 'TRUE' }
VERSION : 0.1
// stored: AutoNumber false, DBAccessibleFromOPCUA true, DBAccessibleFromWebserver true, IsOnlyStoredInLoadMemory false, IsRetainMemResEnabled false, IsWriteProtectedInAS false, MemoryReserve 100
   VAR RETAIN
      "time" : Array[0..32, 0..25] of Int;   // Tiempo de duración de cada paso [modelo, paso]
      number : Array[0..32] of Int;   // Número de pasos por modelo
   END_VAR
   VAR
      stepChangeTimer : DInt := 0;
      stepChangeTimerStart : Bool := FALSE;
      counterDone : Bool := FALSE;
   END_VAR
BEGIN
   "time"[0,0] := 0;
   "time"[0,1..5] := 500;
   "time"[0,6] := 1000;
   "time"[0,7] := 500;
   "time"[0,8] := 1000;
   "time"[0,9..10] := 500;
   "time"[0,11..25] := 0;
   "time"[1,0] := 0;
   "time"[1,1..5] := 500;
   "time"[1,6] := 1000;
   "time"[1,7] := 500;
   "time"[1,8] := 1000;
   "time"[1,9..10] := 500;
   "time"[1,11..25] := 0;
   "time"[2,0] := 0;
   "time"[2,1..5] := 500;
   "time"[2,6] := 1000;
   "time"[2,7] := 500;
   "time"[2,8] := 1000;
   "time"[2,9..10] := 500;
   "time"[2,11..25] := 0;
   "time"[3,0] := 0;
   "time"[3,1] := 500;
   "time"[3,2..4] := 1500;
   "time"[3,5..11] := 500;
   "time"[3,12..25] := 0;
   "time"[4,0] := 0;
   "time"[4,1] := 500;
   "time"[4,2..4] := 1500;
   "time"[4,5..11] := 500;
   "time"[4,12..25] := 0;
   "time"[5,0] := 0;
   "time"[5,1] := 1000;
   "time"[5,2] := 0;
   "time"[5,3] := 1000;
   "time"[5,4..25] := 0;
   "time"[6,0] := 0;
   "time"[6,1..2] := 1500;
   "time"[6,3] := 0;
   "time"[6,4..9] := 3000;
   "time"[6,10..25] := 0;
   "time"[7,0] := 0;
   "time"[7,1..2] := 1500;
   "time"[7,3] := 0;
   "time"[7,4..9] := 3000;
   "time"[7,10..25] := 0;
   "time"[8,0] := 0;
   "time"[8,1..2] := 1500;
   "time"[8,3] := 0;
   "time"[8,4..9] := 3000;
   "time"[8,10..25] := 0;
   "time"[9,0..3] := 0;
   "time"[9,4..5] := 500;
   "time"[9,6..25] := 0;
   "time"[10,0..3] := 0;
   "time"[10,4..5] := 500;
   "time"[10,6..25] := 0;
   "time"[11,0..3] := 0;
   "time"[11,4..5] := 500;
   "time"[11,6..25] := 0;
   "time"[12,0..3] := 0;
   "time"[12,4..5] := 500;
   "time"[12,6..25] := 0;
   "time"[13,0..3] := 0;
   "time"[13,4..5] := 500;
   "time"[13,6..25] := 0;
   "time"[14,0..3] := 0;
   "time"[14,4..5] := 500;
   "time"[14,6..25] := 0;
   "time"[15,0..25] := 0;
   "time"[16,0..3] := 0;
   "time"[16,4..5] := 500;
   "time"[16,6..25] := 0;
   "time"[17,0..3] := 0;
   "time"[17,4..5] := 500;
   "time"[17,6..25] := 0;
   "time"[18,0..3] := 0;
   "time"[18,4..5] := 500;
   "time"[18,6..25] := 0;
   "time"[19,0..3] := 0;
   "time"[19,4..5] := 500;
   "time"[19,6..25] := 0;
   "time"[20,0..25] := 0;
   "time"[21,0..25] := 0;
   "time"[22,0..25] := 0;
   "time"[23,0..25] := 0;
   "time"[24,0..25] := 0;
   "time"[25,0..25] := 0;
   "time"[26,0..25] := 0;
   "time"[27,0..25] := 0;
   "time"[28,0..25] := 0;
   "time"[29,0..25] := 0;
   "time"[30,0..25] := 0;
   "time"[31,0..25] := 0;
   "time"[32,0..25] := 0;
   number[0..2] := 10;
   number[3..4] := 11;
   number[5] := 3;
   number[6..14] := 9;
   number[15] := 8;
   number[16..19] := 9;
   number[20..32] := 0;
END_DATA_BLOCK

DATA_BLOCK "labels"   // DB6
{ S7_Optimized_Access := 'TRUE' }
VERSION : 0.1
// stored: AutoNumber false, DBAccessibleFromOPCUA true, DBAccessibleFromWebserver true, IsOnlyStoredInLoadMemory false, IsRetainMemResEnabled false, IsWriteProtectedInAS false, MemoryReserve 100
   VAR RETAIN
      label1 : Array[0..32] of String[50];   // Etiqueta 1
      label2 : Array[0..32] of String[50];
      label3 : Array[0..32] of String[50];
      label4 : Array[0..32] of String[50];
      label5 : Array[0..32] of String[50];
      label6 : Array[0..32] of String[50];
      posLabel1 : Array[0..32] of Int;   // Posición de etiqueta 1
      posLabel2 : Array[0..32] of Int;
      posLabel3 : Array[0..32] of Int;
      posLabel4 : Array[0..32] of Int;
      posLabel5 : Array[0..32] of Int;
      posLabel6 : Array[0..32] of Int;
      text : Array[0..5] of String;   // Texto HMI de etiquetas
   END_VAR
   VAR
      done2 : Bool := FALSE;
      errorPort2 : Bool := FALSE;
      statusPort2 : Word := 16#7000;
      statusReset : Word := 16#7000;
   END_VAR
   VAR RETAIN
      doneReset : Bool := FALSE;
      scanner1 : Bool := TRUE;
      scanner2 : Bool := TRUE;
      scanner3 : Bool := TRUE;
      scanner4 : Bool := FALSE;
      scanner5 : Bool := FALSE;
   END_VAR
   VAR
      scanner6 : Bool := FALSE;
      scannerOn : Bool := TRUE;
      codeScanned : String := ' ';
      codeReceived : String := '';
      ndr : Bool := FALSE;
      error : Bool := FALSE;
      status : Word := 16#7002;
      lenght : UInt := 0;
      lablelBlock : Array[0..6] of Bool;
      nestScannerRead : String := ' ';
      readScanner : String := '03804073GO23548$R';
      extraction : Array[0..6] of String;
      previousBarcode : String := '';
   END_VAR
BEGIN
   label1[0..4] := '038';
   label1[5] := '1';
   label1[6..8] := '038';
   label1[9] := '202';
   label1[10..11] := '592';
   label1[12] := '202';
   label1[13] := '592';
   label1[14] := '202';
   label1[15..16] := '';
   label1[17] := '592';
   label1[18] := '202';
   label1[19] := '592';
   label1[20..32] := '';
   label2[0..1] := '4066654';
   label2[2] := '4066308';
   label2[3] := '4066654';
   label2[4] := '4066308';
   label2[5] := '2';
   label2[6..7] := '709';
   label2[8] := '706';
   label2[9] := '723';
   label2[10] := '724';
   label2[11] := '723';
   label2[12] := '724';
   label2[13] := '769';
   label2[14] := '768';
   label2[15..16] := '';
   label2[17..18] := '685';
   label2[19] := '163';
   label2[20..32] := '';
   label3[0..1] := '4066430';
   label3[2] := '4066646';
   label3[3] := '4066430';
   label3[4] := '4066646';
   label3[5] := '3';
   label3[6..7] := '708';
   label3[8] := '707';
   label3[9] := '718';
   label3[10] := '719';
   label3[11] := '718';
   label3[12..14] := '719';
   label3[15..16] := '';
   label3[17..18] := '680';
   label3[19] := '161';
   label3[20..32] := '';
   label4[0..32] := '';
   label5[0..32] := '';
   label6[0..32] := '';
   posLabel1[0..14] := 1;
   posLabel1[15..16] := 0;
   posLabel1[17..19] := 1;
   posLabel1[20..32] := 0;
   posLabel2[0..4] := 1;
   posLabel2[5] := 2;
   posLabel2[6..8] := 10;
   posLabel2[9..12] := 5;
   posLabel2[13..14] := 1;
   posLabel2[15..16] := 0;
   posLabel2[17..19] := 5;
   posLabel2[20..32] := 0;
   posLabel3[0..4] := 1;
   posLabel3[5] := 3;
   posLabel3[6..8] := 10;
   posLabel3[9..13] := 5;
   posLabel3[14] := 13;
   posLabel3[15..16] := 0;
   posLabel3[17..19] := 5;
   posLabel3[20..32] := 0;
   posLabel4[0..32] := 0;
   posLabel5[0..32] := 0;
   posLabel6[0..32] := 0;
   text[0] := '';
   text[1] := 'Motor';
   text[2] := 'Track Izq';
   text[3] := 'Track der';
   text[4..5] := '';
   lablelBlock[0] := FALSE;
   lablelBlock[1..3] := TRUE;
   lablelBlock[4..6] := FALSE;
   extraction[0] := '';
   extraction[1] := '038';
   extraction[2..3] := '0380407';
   extraction[4..6] := '';
END_DATA_BLOCK

DATA_BLOCK "conveyor"   // DB41
{ S7_Optimized_Access := 'FALSE' }
VERSION : 0.1
// stored: AutoNumber true, DBAccessibleFromOPCUA true, DBAccessibleFromWebserver true, IsOnlyStoredInLoadMemory false, IsWriteProtectedInAS false
   VAR
      printLabel : Bool := FALSE;
      description : String := 'BACKREST W33A POWER MEMO L6';
      partNumber : String := '2389161X-01';
      lastScann : String := '03804073GO23548$R';
      okModelBit : Bool := FALSE;
      leftTrackScan : String := '4066654X016PN4O385$R';
      rightTrackScan : String := '4066430X016LN4S161$R';
      motorScan : String := '03804073GO23548$R';
   END_VAR
BEGIN
END_DATA_BLOCK

DATA_BLOCK "dataLogging"   // DB36
{ S7_Optimized_Access := 'TRUE' }
VERSION : 0.1
// stored: AutoNumber true, DBAccessibleFromOPCUA true, DBAccessibleFromWebserver true, IsOnlyStoredInLoadMemory false, IsRetainMemResEnabled false, IsWriteProtectedInAS false, MemoryReserve 100
   VAR
      scanning : Array[1..3] of String;
      alignment : Real := 0.0;
      pieceOk : Bool := FALSE;
   END_VAR
BEGIN
   scanning[1] := '03804073GO23548$R';
   scanning[2] := '4066654X016PN4O385$R';
   scanning[3] := '4066430X016LN4S161$R';
END_DATA_BLOCK

DATA_BLOCK "DB_PrinterReference"   // DB33
{ S7_Optimized_Access := 'TRUE' }
VERSION : 0.1
// stored: AutoNumber true, DBAccessibleFromOPCUA true, DBAccessibleFromWebserver true, IsOnlyStoredInLoadMemory false, IsRetainMemResEnabled false, IsWriteProtectedInAS false, MemoryReserve 100
   VAR
      reference : Array[0..32] of "udt_referenceMainInfo";
   END_VAR
BEGIN
   reference[0..32].id := 0;
   reference[0..32].description := '';
   reference[0..32].partNumber := '';
   reference[0..32].rev := '';
   reference[0..32].customerNumber := '';
   reference[0..32].vpps := '';
   reference[0..32].locationCode := '';
   reference[0..32].dataIdentifier := '';
   reference[0..32].duns := '';
END_DATA_BLOCK

DATA_BLOCK "devicesAlarm"   // DB37
{ S7_Optimized_Access := 'TRUE' }
VERSION : 0.1
// stored: AutoNumber true, DBAccessibleFromOPCUA true, DBAccessibleFromWebserver true, IsOnlyStoredInLoadMemory false, IsRetainMemResEnabled false, IsWriteProtectedInAS false, MemoryReserve 100
   VAR
      bannerStatus : Array[0..1023] of Bool;
      manifold : Array[0..1023] of Bool;
      iolink1 : Array[0..1023] of Bool;
      profinetIO1 : Array[0..1023] of Bool;
      profinetIO2 : Array[0..1023] of Bool;
      profinetIO3 : Array[0..1023] of Bool;
      printer : Array[0..1023] of Bool;
      printerDiag : DIS;
   END_VAR
BEGIN
   bannerStatus[0..1023] := FALSE;
   manifold[0..1023] := FALSE;
   iolink1[0..1023] := FALSE;
   profinetIO1[0..1023] := FALSE;
   profinetIO2[0..1023] := FALSE;
   profinetIO3[0..1023] := FALSE;
   printer[0..1023] := FALSE;
   printerDiag.MaintainanceState := 16#0000_0000;
   printerDiag.ComponentStateDetail := 16#0000_8000;
   printerDiag.OwnState := 0;
   printerDiag.IOState := 16#0001;
   printerDiag.OperatingState := 0;
END_DATA_BLOCK

DATA_BLOCK "hmi"   // DB7
{ S7_Optimized_Access := 'TRUE' }
VERSION : 0.1
// stored: AutoNumber true, DBAccessibleFromOPCUA true, DBAccessibleFromWebserver true, IsOnlyStoredInLoadMemory false, IsRetainMemResEnabled false, IsWriteProtectedInAS false, MemoryReserve 100
   VAR
      modeButton : Bool := FALSE;
      mode : Int := 2;
      model : Array[0..32] of Bool;
      recipeStep : Int := 9;
      "a" : DInt := 44690590;
      "b" : DInt := 536_871_082;
      mascA : DInt := 66846862;
      mascB : DInt := 0;
      recipeStepTime : Int := 500;
      recipeStepSubstract : Bool := FALSE;
      recipeStepAdd : Bool := FALSE;
      recipeLastStep : Int := 9;
      updateStep : Bool := FALSE;
      moveToCurrentStep : Bool := FALSE;
      recordA1 : Bool := FALSE;
      readA1 : Bool := FALSE;
      recordA2 : Bool := FALSE;
      readA2 : Bool := FALSE;
      recordB1 : Bool := FALSE;
      readB1 : Bool := FALSE;
      recordB2 : Bool := FALSE;
      readB2 : Bool := FALSE;
      recordAnalog : Bool := FALSE;
      readAnalog : Bool := FALSE;
      recipeStepQuantity : Int := 10;
      eraseStep : Bool := FALSE;
      insertStep : Bool := FALSE;
      copyStep : Bool := FALSE;
      copySequence : Bool := FALSE;
      copySequenceStep : Bool := FALSE;
      baseStep : Int := 10;
      destinationStep : Int := 11;
      baseModel : Int := 7;
      destinationModel : Int := 8;
      baseModelStep : Int := 0;
      modelDestinationStep : Int := 0;
      baseModelStep_1 : Int := 2;
      modelDestinationStep_1 : Int := 3;
      operatorTextIndicator : String := ' ';
      enableStationAir : Bool := FALSE;
      enableAirHmiPermission : Bool := FALSE;
      insertAlarmKey : Bool := FALSE;
      enableStationVisualizationButton : Bool := FALSE;
      enableStationHideAlarmButton : Bool := FALSE;
      alarmAckmowledge : Bool := FALSE;
      home : Bool := FALSE;
      advancePercentage : Real := 0.0;
      administratorAlarmButton : Bool := FALSE;
      activateLamp : Bool := FALSE;
      activateFan : Bool := TRUE;
   END_VAR
   VAR RETAIN
      cicles : Int := 444;
      production1 : Int := 80;
      production2 : Int := 48;
      production3 : Int := 17;
   END_VAR
   VAR
      productionRestart1 : Bool := FALSE;
      productionRestart2 : Bool := FALSE;
      productionRestart3 : Bool := FALSE;
      cyclesRestart : Bool := FALSE;
      manualPrint : Bool := FALSE;
      BLOQUEO : Bool := TRUE;
      manualModeNecessary : Bool := FALSE;
      modelChange : Bool := FALSE;
      alarmManualButton : Bool := FALSE;
      user : String := 'Administrator';
      pass : String := 'PASSWORD';
   END_VAR
BEGIN
   model[0..32] := FALSE;
END_DATA_BLOCK

DATA_BLOCK "sensorDistribution"   // DB129
{ S7_Optimized_Access := 'TRUE' }
VERSION : 0.1
// stored: AutoNumber false, DBAccessibleFromOPCUA true, DBAccessibleFromWebserver true, IsOnlyStoredInLoadMemory false, IsRetainMemResEnabled false, IsWriteProtectedInAS false, MemoryReserve 100
   VAR
      inputsStatus : Array[0..31] of Byte;
      outputsStatus : Array[0..31] of Byte;
   END_VAR
BEGIN
   inputsStatus[0..5] := 16#00;
   inputsStatus[6] := 16#01;
   inputsStatus[7] := 16#00;
   inputsStatus[8] := 16#01;
   inputsStatus[9..16] := 16#00;
   inputsStatus[17..18] := 16#01;
   inputsStatus[19..31] := 16#00;
   outputsStatus[0] := 16#01;
   outputsStatus[1] := 16#00;
   outputsStatus[2] := 16#01;
   outputsStatus[3] := 16#00;
   outputsStatus[4] := 16#01;
   outputsStatus[5] := 16#00;
   outputsStatus[6] := 16#01;
   outputsStatus[7..31] := 16#00;
END_DATA_BLOCK

DATA_BLOCK "inputs"   // DB1
{ S7_Optimized_Access := 'TRUE' }
VERSION : 0.1
// stored: AutoNumber false, DBAccessibleFromOPCUA true, DBAccessibleFromWebserver true, IsOnlyStoredInLoadMemory false, IsRetainMemResEnabled false, IsWriteProtectedInAS false, MemoryReserve 100
   VAR RETAIN
      inputSequence : Array[0..32, 0..25] of DInt;   // 32 entradas [modelo, paso]
   END_VAR
   VAR
      activeInputsReq : Array[0..31] of Bool;
   END_VAR
   VAR RETAIN
      maskSequence : Array[0..32, 0..25] of DInt;   // Máscara de entradas
   END_VAR
   VAR
      activeMask : Array[0..31] of Bool;
   END_VAR
   VAR RETAIN
      inputText : Array[0..31] of String;   // Texto HMI de cada entrada
   END_VAR
   VAR
      buttonStatus : Array[0..63] of Bool;
      activeInputsReqDInt : DInt := 131392;   // Estado de sensores en directo
      inputActive : Array[0..31] of Bool;
      euchnerReading : Array[0..254] of Char;
      nestScannerReading : String := '';
      upperScannerReading : String := '';
      nestScanerReceived : Array[0..254] of Char;
      nestScanerReceivedString : String := '';
      upperScannerReceived : Array[0..254] of Char;
      upperScannerReceivedString : String := '';
      euchnerReadingString : String := '$01';
      laserReading : Word := 16#0000;
      laserConstant : Real := 0.0005802801;
      laserReadingInt : DInt := 0;
      readingConversion : LReal := 0.0;
      euchnerName : String := '';
      euchner : Array[0..257] of Byte;
   END_VAR
BEGIN
   inputSequence[0,0] := 23724353;
   inputSequence[0,1] := 827_518_278;
   inputSequence[0,2..4] := 44756294;
   inputSequence[0,5] := 1_252_650_334;
   inputSequence[0,6..7] := 1_118_432_670;
   inputSequence[0,8] := 1_118_432_414;
   inputSequence[0,9] := 44690590;
   inputSequence[0,10] := 44892160;
   inputSequence[0,11..25] := 0;
   inputSequence[1,0] := 23724353;
   inputSequence[1,1] := 827_518_278;
   inputSequence[1,2..4] := 44756294;
   inputSequence[1,5] := 1_252_650_334;
   inputSequence[1,6..7] := 1_118_432_670;
   inputSequence[1,8] := 1_118_432_414;
   inputSequence[1,9] := 44690590;
   inputSequence[1,10] := 44892160;
   inputSequence[1,11..25] := 0;
   inputSequence[2,0] := 23724353;
   inputSequence[2,1] := 827_514_182;
   inputSequence[2,2..4] := 44752198;
   inputSequence[2,5] := 1_252_646_238;
   inputSequence[2,6..7] := 1_118_428_574;
   inputSequence[2,8] := 1_118_428_318;
   inputSequence[2,9] := 44686494;
   inputSequence[2,10] := 44892160;
   inputSequence[2,11..25] := 0;
   inputSequence[3,0] := 23724353;
   inputSequence[3,1] := 827_518_278;
   inputSequence[3,2..4] := 44756294;
   inputSequence[3,5] := 1_252_650_334;
   inputSequence[3,6..8] := 1_118_432_670;
   inputSequence[3,9] := 1_118_432_414;
   inputSequence[3,10] := 44690590;
   inputSequence[3,11] := 44892160;
   inputSequence[3,12..25] := 0;
   inputSequence[4,0] := 23724353;
   inputSequence[4,1] := 827_514_182;
   inputSequence[4,2..4] := 44752198;
   inputSequence[4,5] := 1_252_646_238;
   inputSequence[4,6..7] := 1_118_428_574;
   inputSequence[4,8] := 1_118_428_446;
   inputSequence[4,9] := 1_118_428_318;
   inputSequence[4,10] := 44686494;
   inputSequence[4,11] := 44892160;
   inputSequence[4,12..25] := 0;
   inputSequence[5,0..1] := 64;
   inputSequence[5,2..3] := 128;
   inputSequence[5,4..25] := 0;
   inputSequence[6,0] := 23724353;
   inputSequence[6,1] := 827_780_422;
   inputSequence[6,2] := 44756294;
   inputSequence[6,3] := 44755974;
   inputSequence[6,4] := 1_252_650_334;
   inputSequence[6,5..7] := 1_118_432_670;
   inputSequence[6,8] := 1_118_432_414;
   inputSequence[6,9] := 44630336;
   inputSequence[6,10..25] := 0;
   inputSequence[7,0] := 23724353;
   inputSequence[7,1] := 827_780_422;
   inputSequence[7,2] := 44756294;
   inputSequence[7,3] := 44755974;
   inputSequence[7,4] := 1_252_650_334;
   inputSequence[7,5..7] := 1_118_432_670;
   inputSequence[7,8] := 1_118_432_414;
   inputSequence[7,9] := 44630336;
   inputSequence[7,10..25] := 0;
   inputSequence[8,0] := 23724353;
   inputSequence[8,1] := 827_776_326;
   inputSequence[8,2] := 44752198;
   inputSequence[8,3] := 44751878;
   inputSequence[8,4] := 1_252_646_238;
   inputSequence[8,5] := 1_118_428_574;
   inputSequence[8,6] := 1_118_428_318;
   inputSequence[8,7] := 1_118_428_574;
   inputSequence[8,8] := 1_118_428_318;
   inputSequence[8,9] := 44630336;
   inputSequence[8,10..25] := 0;
   inputSequence[9,0] := 321;
   inputSequence[9,1] := 4193656;
   inputSequence[9,2] := 2_017_459_576;
   inputSequence[9,3] := 1_077_935_482;
   inputSequence[9,4] := 1_073_745_282;
   inputSequence[9,5..6] := 1_073_745_538;
   inputSequence[9,7..9] := 320;
   inputSequence[9,10..25] := 0;
   inputSequence[10,0] := 321;
   inputSequence[10,1] := 4193656;
   inputSequence[10,2] := 2_017_459_576;
   inputSequence[10,3] := 1_077_935_482;
   inputSequence[10,4] := 1_073_745_282;
   inputSequence[10,5..6] := 1_073_745_538;
   inputSequence[10,7..9] := 320;
   inputSequence[10,10..25] := 0;
   inputSequence[11,0] := 321;
   inputSequence[11,1] := 4193656;
   inputSequence[11,2] := 2_017_459_576;
   inputSequence[11,3] := 1_077_935_482;
   inputSequence[11,4] := 1_073_745_282;
   inputSequence[11,5..6] := 1_073_745_538;
   inputSequence[11,7..9] := 320;
   inputSequence[11,10..25] := 0;
   inputSequence[12,0] := 321;
   inputSequence[12,1] := 8387960;
   inputSequence[12,2] := 2_021_653_880;
   inputSequence[12,3] := 1_082_129_786;
   inputSequence[12,4] := 1_077_939_586;
   inputSequence[12,5] := 1_077_939_842;
   inputSequence[12,6] := 1_073_745_538;
   inputSequence[12,7..9] := 320;
   inputSequence[12,10..25] := 0;
   inputSequence[13,0] := 321;
   inputSequence[13,1] := 4193656;
   inputSequence[13,2] := 2_017_459_576;
   inputSequence[13,3] := 1_077_935_482;
   inputSequence[13,4] := 1_073_745_282;
   inputSequence[13,5..6] := 1_073_745_538;
   inputSequence[13,7..9] := 320;
   inputSequence[13,10..25] := 0;
   inputSequence[14,0] := 321;
   inputSequence[14,1] := 4193656;
   inputSequence[14,2] := 2_017_459_576;
   inputSequence[14,3] := 1_077_935_482;
   inputSequence[14,4] := 1_073_745_282;
   inputSequence[14,5..6] := 1_073_745_538;
   inputSequence[14,7..9] := 320;
   inputSequence[14,10..25] := 0;
   inputSequence[15,0] := 11;
   inputSequence[15,1] := 63040522;
   inputSequence[15,2] := 1_338_108_938;
   inputSequence[15,3] := 65137674;
   inputSequence[15,4] := 65135628;
   inputSequence[15,5] := 65134612;
   inputSequence[15,6] := 57344;
   inputSequence[15,7] := 805_363_712;
   inputSequence[15,8] := 10;
   inputSequence[15,9..25] := 0;
   inputSequence[16,0] := 321;
   inputSequence[16,1] := 8387960;
   inputSequence[16,2] := 2_021_653_880;
   inputSequence[16,3] := 1_082_129_786;
   inputSequence[16,4] := 1_077_939_586;
   inputSequence[16,5] := 1_077_939_842;
   inputSequence[16,6] := 1_073_745_538;
   inputSequence[16,7..9] := 320;
   inputSequence[16,10..25] := 0;
   inputSequence[17,0] := 321;
   inputSequence[17,1] := 4193656;
   inputSequence[17,2] := 2_017_459_576;
   inputSequence[17,3] := 1_077_935_482;
   inputSequence[17,4] := 1_073_745_282;
   inputSequence[17,5..6] := 1_073_745_538;
   inputSequence[17,7..9] := 320;
   inputSequence[17,10..25] := 0;
   inputSequence[18,0] := 321;
   inputSequence[18,1] := 4193656;
   inputSequence[18,2] := 2_017_459_576;
   inputSequence[18,3] := 1_077_935_482;
   inputSequence[18,4] := 1_073_745_282;
   inputSequence[18,5..6] := 1_073_745_538;
   inputSequence[18,7..9] := 320;
   inputSequence[18,10..25] := 0;
   inputSequence[19,0] := 321;
   inputSequence[19,1] := 4193656;
   inputSequence[19,2] := 2_017_459_576;
   inputSequence[19,3] := 1_077_935_482;
   inputSequence[19,4] := 1_073_745_282;
   inputSequence[19,5..6] := 1_073_745_538;
   inputSequence[19,7..9] := 320;
   inputSequence[19,10..25] := 0;
   inputSequence[20,0..25] := 0;
   inputSequence[21,0..25] := 0;
   inputSequence[22,0..25] := 0;
   inputSequence[23,0..25] := 0;
   inputSequence[24,0..25] := 0;
   inputSequence[25,0..25] := 0;
   inputSequence[26,0..25] := 0;
   inputSequence[27,0..25] := 0;
   inputSequence[28,0..25] := 0;
   inputSequence[29,0..25] := 0;
   inputSequence[30,0..25] := 0;
   inputSequence[31,0..25] := 0;
   inputSequence[32,0..25] := 0;
   activeInputsReq[0] := TRUE;
   activeInputsReq[1..5] := FALSE;
   activeInputsReq[6] := TRUE;
   activeInputsReq[7] := FALSE;
   activeInputsReq[8] := TRUE;
   activeInputsReq[9..16] := FALSE;
   activeInputsReq[17] := TRUE;
   activeInputsReq[18] := FALSE;
   activeInputsReq[19] := TRUE;
   activeInputsReq[20] := FALSE;
   activeInputsReq[21..22] := TRUE;
   activeInputsReq[23] := FALSE;
   activeInputsReq[24] := TRUE;
   activeInputsReq[25..31] := FALSE;
   maskSequence[0,0] := 66859008;
   maskSequence[0,1] := 66846720;
   maskSequence[0,2] := 66847168;
   maskSequence[0,3..4] := 66846848;
   maskSequence[0,5..8] := 66846720;
   maskSequence[0,9] := 66846862;
   maskSequence[0,10] := 66649232;
   maskSequence[0,11..25] := 0;
   maskSequence[1,0] := 66859008;
   maskSequence[1,1] := 66846720;
   maskSequence[1,2] := 66847168;
   maskSequence[1,3..4] := 66846848;
   maskSequence[1,5..8] := 66846720;
   maskSequence[1,9] := 66846862;
   maskSequence[1,10] := 66649232;
   maskSequence[1,11..25] := 0;
   maskSequence[2,0] := 66859008;
   maskSequence[2,1] := 66846720;
   maskSequence[2,2] := 66847168;
   maskSequence[2,3..4] := 66846848;
   maskSequence[2,5..8] := 66846720;
   maskSequence[2,9] := 66846862;
   maskSequence[2,10] := 66649232;
   maskSequence[2,11..25] := 0;
   maskSequence[3,0] := 66859008;
   maskSequence[3,1] := 66846720;
   maskSequence[3,2] := 66847168;
   maskSequence[3,3..4] := 66846848;
   maskSequence[3,5..7] := 66846720;
   maskSequence[3,8] := 66846976;
   maskSequence[3,9] := 66846720;
   maskSequence[3,10] := 66846848;
   maskSequence[3,11] := 66649232;
   maskSequence[3,12..25] := 0;
   maskSequence[4,0] := 66859008;
   maskSequence[4,1] := 66846720;
   maskSequence[4,2] := 66847168;
   maskSequence[4,3..4] := 66846848;
   maskSequence[4,5..7] := 66846720;
   maskSequence[4,8] := 66847168;
   maskSequence[4,9] := 66846720;
   maskSequence[4,10] := 66846848;
   maskSequence[4,11] := 66649232;
   maskSequence[4,12..25] := 0;
   maskSequence[5,0..1] := -65;
   maskSequence[5,2..3] := -129;
   maskSequence[5,4..25] := 0;
   maskSequence[6,0..2] := 66846720;
   maskSequence[6,3] := 66847168;
   maskSequence[6,4..8] := 66846720;
   maskSequence[6,9] := 66847168;
   maskSequence[6,10..25] := 0;
   maskSequence[7,0..1] := 66846720;
   maskSequence[7,2..3] := 66847168;
   maskSequence[7,4..6] := 66846720;
   maskSequence[7,7] := 66846976;
   maskSequence[7,8] := 66846720;
   maskSequence[7,9] := 66847168;
   maskSequence[7,10..25] := 0;
   maskSequence[8,0..1] := 66846720;
   maskSequence[8,2..3] := 66847168;
   maskSequence[8,4..5] := 66846720;
   maskSequence[8,6..7] := 66846976;
   maskSequence[8,8] := 66846720;
   maskSequence[8,9] := 66847168;
   maskSequence[8,10..25] := 0;
   maskSequence[9,0] := -322;
   maskSequence[9,1] := 2_014_248_960;
   maskSequence[9,2..3] := 983040;
   maskSequence[9,4..5] := 79687736;
   maskSequence[9,6] := 134_213_948;
   maskSequence[9,7..8] := -2;
   maskSequence[9,9] := 134_217_406;
   maskSequence[9,10..25] := 0;
   maskSequence[10,0] := -322;
   maskSequence[10,1] := 2_014_289_920;
   maskSequence[10,2..3] := 1024000;
   maskSequence[10,4..5] := 79687736;
   maskSequence[10,6] := 134_213_948;
   maskSequence[10,7..8] := -2;
   maskSequence[10,9] := 134_217_406;
   maskSequence[10,10..25] := 0;
   maskSequence[11,0] := -322;
   maskSequence[11,1] := 2_014_248_960;
   maskSequence[11,2..3] := 983040;
   maskSequence[11,4..5] := 79687736;
   maskSequence[11,6] := 134_213_948;
   maskSequence[11,7..8] := -2;
   maskSequence[11,9] := 134_217_406;
   maskSequence[11,10..25] := 0;
   maskSequence[12,0] := -322;
   maskSequence[12,1] := 2_014_248_960;
   maskSequence[12,2..3] := 983040;
   maskSequence[12,4..5] := 79687736;
   maskSequence[12,6] := 134_213_948;
   maskSequence[12,7..8] := -2;
   maskSequence[12,9] := 134_217_406;
   maskSequence[12,10..25] := 0;
   maskSequence[13,0] := -322;
   maskSequence[13,1] := 2_014_248_960;
   maskSequence[13,2..3] := 983040;
   maskSequence[13,4..5] := 79687736;
   maskSequence[13,6] := 134_213_948;
   maskSequence[13,7..8] := -2;
   maskSequence[13,9] := 134_217_406;
   maskSequence[13,10..25] := 0;
   maskSequence[14,0] := -322;
   maskSequence[14,1] := 2_014_248_960;
   maskSequence[14,2] := 806_289_408;
   maskSequence[14,3] := 983040;
   maskSequence[14,4..5] := 79687736;
   maskSequence[14,6] := 134_213_948;
   maskSequence[14,7..8] := -2;
   maskSequence[14,9] := 134_217_406;
   maskSequence[14,10..25] := 0;
   maskSequence[15,0] := 0;
   maskSequence[15,1] := 2_080_374_784;
   maskSequence[15,2..3] := 805_306_368;
   maskSequence[15,4..5] := 868_220_928;
   maskSequence[15,6..7] := 268_435_452;
   maskSequence[15,8..25] := 0;
   maskSequence[16,0] := -322;
   maskSequence[16,1] := 2_014_248_960;
   maskSequence[16,2..3] := 983040;
   maskSequence[16,4..5] := 79687736;
   maskSequence[16,6] := 134_213_948;
   maskSequence[16,7..8] := -2;
   maskSequence[16,9] := 134_217_406;
   maskSequence[16,10..25] := 0;
   maskSequence[17,0] := -322;
   maskSequence[17,1] := 2_014_248_960;
   maskSequence[17,2..3] := 983040;
   maskSequence[17,4..5] := 79687736;
   maskSequence[17,6] := 134_213_948;
   maskSequence[17,7..8] := -2;
   maskSequence[17,9] := 134_217_406;
   maskSequence[17,10..25] := 0;
   maskSequence[18,0] := -322;
   maskSequence[18,1] := 2_014_248_960;
   maskSequence[18,2..3] := 983040;
   maskSequence[18,4..5] := 79687736;
   maskSequence[18,6] := 134_213_948;
   maskSequence[18,7..8] := -2;
   maskSequence[18,9] := 134_217_406;
   maskSequence[18,10..25] := 0;
   maskSequence[19,0] := -322;
   maskSequence[19,1] := 2_014_248_960;
   maskSequence[19,2..3] := 983040;
   maskSequence[19,4..5] := 79687736;
   maskSequence[19,6] := 134_213_948;
   maskSequence[19,7..8] := -2;
   maskSequence[19,9] := 134_217_406;
   maskSequence[19,10..25] := 0;
   maskSequence[20,0..25] := 0;
   maskSequence[21,0..25] := 0;
   maskSequence[22,0..25] := 0;
   maskSequence[23,0..25] := 0;
   maskSequence[24,0..25] := 0;
   maskSequence[25,0..25] := 0;
   maskSequence[26,0..25] := 0;
   maskSequence[27,0..25] := 0;
   maskSequence[28,0..25] := 0;
   maskSequence[29,0..25] := 0;
   maskSequence[30,0..25] := 0;
   maskSequence[31,0..25] := 0;
   maskSequence[32,0..25] := 0;
   activeMask[0..11] := FALSE;
   activeMask[12..13] := TRUE;
   activeMask[14..17] := FALSE;
   activeMask[18..25] := TRUE;
   activeMask[26..31] := FALSE;
   inputText[0] := 'CLEAR DATA';
   inputText[1] := 'Clamp izq. cerrado PRX18151';
   inputText[2] := 'Clamp der. cerrado PRX18150';
   inputText[3] := 'Clamp plastic bridge cerrado PRX19130';
   inputText[4] := 'Plastic bridge presente PRX19090';
   inputText[5] := 'Reserva';
   inputText[6] := 'Herramental izq. pos. inicio PRX18130';
   inputText[7] := 'Herramental izq pos trabajo PRX19091';
   inputText[8] := 'Herramental der. pos. inicio PRX18131';
   inputText[9] := 'Reserva';
   inputText[10] := 'Track 1 izq. presente PRX18090';
   inputText[11] := 'Track 1 der. presente PRX18110';
   inputText[12] := 'Tornillo track izq. PRX19110';
   inputText[13] := 'Tornillo track der. PRX19111';
   inputText[14] := 'Track 2 izq. presente PRX18091';
   inputText[15] := 'Track 2 der. presente PRX18111';
   inputText[16] := 'Posicion nido colocar track PRX19150';
   inputText[17] := 'Posicion nido ensamble varilla PRX19151';
   inputText[18] := 'Quitar pieza';
   inputText[19..26] := 'Reserva';
   inputText[27] := 'Escaner motor OK';
   inputText[28] := 'Escaner Track izq OK';
   inputText[29] := 'Escaner Track der OK';
   inputText[30] := 'Motor conectado ';
   inputText[31] := 'RESERVA';
   buttonStatus[0] := FALSE;
   buttonStatus[1..4] := TRUE;
   buttonStatus[5..6] := FALSE;
   buttonStatus[7] := TRUE;
   buttonStatus[8..9] := FALSE;
   buttonStatus[10..11] := TRUE;
   buttonStatus[12] := FALSE;
   buttonStatus[13..16] := TRUE;
   buttonStatus[17..18] := FALSE;
   buttonStatus[19] := TRUE;
   buttonStatus[20] := FALSE;
   buttonStatus[21] := TRUE;
   buttonStatus[22] := FALSE;
   buttonStatus[23] := TRUE;
   buttonStatus[24] := FALSE;
   buttonStatus[25] := TRUE;
   buttonStatus[26..32] := FALSE;
   buttonStatus[33..35] := TRUE;
   buttonStatus[36..38] := FALSE;
   buttonStatus[39] := TRUE;
   buttonStatus[40..49] := FALSE;
   buttonStatus[50..57] := TRUE;
   buttonStatus[58..63] := FALSE;
   inputActive[0..5] := FALSE;
   inputActive[6] := TRUE;
   inputActive[7] := FALSE;
   inputActive[8] := TRUE;
   inputActive[9..16] := FALSE;
   inputActive[17..18] := TRUE;
   inputActive[19..31] := FALSE;
   euchnerReading[0] := '$01';
   euchnerReading[1..127] := '$00';
   euchnerReading[128..254] := ' ';
   nestScanerReceived[0..254] := ' ';
   upperScannerReceived[0..254] := ' ';
   euchner[0..1] := 16#00;
   euchner[2] := 16#44;
   euchner[3..7] := 16#00;
   euchner[8..147] := 16#20;
   euchner[148..257] := 16#00;
END_DATA_BLOCK

DATA_BLOCK "outputs"   // DB2
{ S7_Optimized_Access := 'TRUE' }
VERSION : 0.1
// stored: AutoNumber false, DBAccessibleFromOPCUA true, DBAccessibleFromWebserver true, IsOnlyStoredInLoadMemory false, IsRetainMemResEnabled false, IsWriteProtectedInAS false, MemoryReserve 0
   VAR RETAIN
      outputSequence : Array[0..32, 0..25] of DInt;   // 32 salidas [modelo, paso]
   END_VAR
   VAR
      activeOutputsReq : Array[0..31] of Bool;
   END_VAR
   VAR RETAIN
      maskSequence : Array[0..32, 0..25] of DInt;   // Máscara de salidas
   END_VAR
   VAR
      activeMask : Array[0..31] of Bool;
      active : DInt := 85;
      outputsActive : Array[0..31] of Bool;
   END_VAR
   VAR RETAIN
      text : Array[0..31] of String;   // Texto HMI de cada salida
   END_VAR
   VAR
      availableNameManipulate : Array[0..8] of String;   // Texto HMI en pagina Manual
      status : Array[0..63] of Bool;
      cylinderDirectionA : Array[0..9] of Bool;   // Variable HMI para activar avance
      cylinderDirectionB : Array[0..9] of Bool;   // Variable HMI para activar retroceso
      cylinderDirectionAActive : Array[0..9] of Bool;   // Variable HMI para enclavamiento avance
      cylinderDirectionBActive : Array[0..9] of Bool;   // Variable HMI para enclavamiento retroceso
      cylinderDirectionAStatus : Array[0..9] of Bool;   // Variable HMI para enclavamiento avance
      cylinderDirectionBStatus : Array[0..9] of Bool;   // Variable HMI para enclavamiento retroceso
      vent : Array[0..9] of Bool;   // Variable HMI para desactivar electroválvula
      cylinderStatus : Array[0..9] of Int;   // Variable HMI para estado de los botones de manipulación
      activateOutput : Array[0..31] of Bool;
      activeAlarm : Bool := FALSE;
      showTextsOutputs : Bool := FALSE;
      cicleTime : Int := 0;
      cicleTimeTimerReset : Bool := FALSE;
      timer1 { S7_SetPoint := 'True'} : TON_TIME;
      timer2 { S7_SetPoint := 'True'} : TON_TIME;
      timer3 { S7_SetPoint := 'True'} : TON_TIME;
      timer4 { S7_SetPoint := 'True'} : TON_TIME;
      timer5 { S7_SetPoint := 'True'} : TON_TIME;
      timer6 { S7_SetPoint := 'True'} : TON_TIME;
      timer7 { S7_SetPoint := 'True'} : TON_TIME;
      timer8 { S7_SetPoint := 'True'} : TON_TIME;
      timer9 { S7_SetPoint := 'True'} : TON_TIME;
      timer10 { S7_SetPoint := 'True'} : TON_TIME;
      timer11 { S7_SetPoint := 'True'} : TON_TIME;
      timer12 { S7_SetPoint := 'True'} : TON_TIME;
      timer13 { S7_SetPoint := 'True'} : TON_TIME;
      timer14 { S7_SetPoint := 'True'} : TON_TIME;
      timer15 { S7_SetPoint := 'True'} : TON_TIME;
      timer16 { S7_SetPoint := 'True'} : TON_TIME;
      timer17 { S7_SetPoint := 'True'} : TON_TIME;
      timer18 { S7_SetPoint := 'True'} : TON_TIME;
      timer19 { S7_SetPoint := 'True'} : TON_TIME;
      timer20 { S7_SetPoint := 'True'} : TON_TIME;
      timer21 { S7_SetPoint := 'True'} : TON_TIME;
      timer22 { S7_SetPoint := 'True'} : TON_TIME;
      timer23 { S7_SetPoint := 'True'} : TON_TIME;
      timer24 { S7_SetPoint := 'True'} : TON_TIME;
      timer25 { S7_SetPoint := 'True'} : TON_TIME;
      timer26 { S7_SetPoint := 'True'} : TON_TIME;
      timer27 { S7_SetPoint := 'True'} : TON_TIME;
      timer28 { S7_SetPoint := 'True'} : TON_TIME;
      timer29 { S7_SetPoint := 'True'} : TON_TIME;
      timer30 { S7_SetPoint := 'True'} : TON_TIME;
      timer31 { S7_SetPoint := 'True'} : TON_TIME;
      "timer" { S7_SetPoint := 'True'} : Array[0..31] of ton_time;
      reset : Bool := FALSE;
      timerReset : Bool := FALSE;
      visibility : Array[0..8] of Bool;
      visualizeCicleTime : Int := 111;
      energysaverTimer { S7_SetPoint := 'True'} : TON_TIME;
      scannerOk : Array[0..5] of Bool;
      scannerLength : Array[0..5] of Int;
      cilinder1 : Bool := TRUE;
      cilinder2 : Bool := TRUE;
      cilinder3 : Bool := TRUE;
      cilinder4 : Bool := FALSE;
      cilinder5 : Bool := FALSE;
      cilinder6 : Bool := FALSE;
      cilinder7 : Bool := FALSE;
      cilinder8 : Bool := FALSE;
   END_VAR
BEGIN
   outputSequence[0,0] := 90;
   outputSequence[0,1] := 85;
   outputSequence[0,2] := 166;
   outputSequence[0,3] := 422;
   outputSequence[0,4] := 681;
   outputSequence[0,5] := 165;
   outputSequence[0,6] := 66726;
   outputSequence[0,7] := 170;
   outputSequence[0,8] := 133289;
   outputSequence[0,9] := 536_871_082;
   outputSequence[0,10] := 90;
   outputSequence[0,11..25] := 0;
   outputSequence[1,0] := 90;
   outputSequence[1,1] := 85;
   outputSequence[1,2] := 166;
   outputSequence[1,3] := 422;
   outputSequence[1,4] := 681;
   outputSequence[1,5] := 165;
   outputSequence[1,6] := 66726;
   outputSequence[1,7] := 170;
   outputSequence[1,8] := 133289;
   outputSequence[1,9] := 536_871_082;
   outputSequence[1,10] := 90;
   outputSequence[1,11..25] := 0;
   outputSequence[2,0] := 90;
   outputSequence[2,1] := 85;
   outputSequence[2,2] := 166;
   outputSequence[2,3] := 422;
   outputSequence[2,4] := 681;
   outputSequence[2,5] := 165;
   outputSequence[2,6] := 66726;
   outputSequence[2,7] := 170;
   outputSequence[2,8] := 133289;
   outputSequence[2,9] := 536_871_082;
   outputSequence[2,10] := 90;
   outputSequence[2,11..25] := 0;
   outputSequence[3,0] := 90;
   outputSequence[3,1] := 85;
   outputSequence[3,2] := 170;
   outputSequence[3,3] := 938;
   outputSequence[3,4] := 170;
   outputSequence[3,5] := 1194;
   outputSequence[3,6..7] := 1193;
   outputSequence[3,8] := 3241;
   outputSequence[3,9] := 80;
   outputSequence[3,10] := 90;
   outputSequence[3,11..25] := 0;
   outputSequence[4,0] := -1_073_741_488;
   outputSequence[4,1] := -956_301_013;
   outputSequence[4,2] := 117_440_810;
   outputSequence[4,3] := -1_073_741_653;
   outputSequence[4,4] := 65715;
   outputSequence[4,5] := 65739;
   outputSequence[4,6] := 171;
   outputSequence[4,7] := 301;
   outputSequence[4,8] := 134_742_317;
   outputSequence[4,9] := 341;
   outputSequence[4,10..25] := 0;
   outputSequence[5,0] := 90;
   outputSequence[5,1] := 89;
   outputSequence[5,2] := 90;
   outputSequence[5,3] := 89;
   outputSequence[5,4..25] := 0;
   outputSequence[6,0] := 90;
   outputSequence[6,1] := 85;
   outputSequence[6,2] := 170;
   outputSequence[6,3] := 938;
   outputSequence[6,4] := 170;
   outputSequence[6,5] := 66730;
   outputSequence[6,6] := 170;
   outputSequence[6,7] := 169;
   outputSequence[6,8] := 133289;
   outputSequence[6,9] := 89;
   outputSequence[6,10..25] := 0;
   outputSequence[7,0] := 90;
   outputSequence[7,1] := 85;
   outputSequence[7,2] := 170;
   outputSequence[7,3] := 938;
   outputSequence[7,4] := 170;
   outputSequence[7,5] := 66726;
   outputSequence[7,6] := 170;
   outputSequence[7,7] := 169;
   outputSequence[7,8] := 133289;
   outputSequence[7,9] := 89;
   outputSequence[7,10..25] := 0;
   outputSequence[8,0] := 90;
   outputSequence[8,1] := 85;
   outputSequence[8,2] := 170;
   outputSequence[8,3] := 938;
   outputSequence[8,4] := 170;
   outputSequence[8,5] := 66726;
   outputSequence[8,6] := 170;
   outputSequence[8,7] := 169;
   outputSequence[8,8] := 133289;
   outputSequence[8,9] := 89;
   outputSequence[8,10..25] := 0;
   outputSequence[9,0] := 336;
   outputSequence[9,1] := 298;
   outputSequence[9,2] := 299;
   outputSequence[9,3] := 171;
   outputSequence[9,4] := 65715;
   outputSequence[9,5] := 65739;
   outputSequence[9,6] := 171;
   outputSequence[9,7] := 301;
   outputSequence[9,8] := 134_742_317;
   outputSequence[9,9] := 341;
   outputSequence[9,10..25] := 0;
   outputSequence[10,0] := 336;
   outputSequence[10,1] := 298;
   outputSequence[10,2] := 299;
   outputSequence[10,3] := 171;
   outputSequence[10,4] := 65715;
   outputSequence[10,5] := 65739;
   outputSequence[10,6] := 171;
   outputSequence[10,7] := 301;
   outputSequence[10,8] := 134_742_317;
   outputSequence[10,9] := 341;
   outputSequence[10,10..25] := 0;
   outputSequence[11,0] := 336;
   outputSequence[11,1] := 298;
   outputSequence[11,2] := 299;
   outputSequence[11,3] := 171;
   outputSequence[11,4] := 65715;
   outputSequence[11,5] := 65739;
   outputSequence[11,6] := 171;
   outputSequence[11,7] := 301;
   outputSequence[11,8] := 134_742_317;
   outputSequence[11,9] := 341;
   outputSequence[11,10..25] := 0;
   outputSequence[12,0] := 336;
   outputSequence[12,1] := 298;
   outputSequence[12,2] := 299;
   outputSequence[12,3] := 171;
   outputSequence[12,4] := 65715;
   outputSequence[12,5] := 65739;
   outputSequence[12,6] := 171;
   outputSequence[12,7] := 301;
   outputSequence[12,8] := 134_742_317;
   outputSequence[12,9] := 341;
   outputSequence[12,10..25] := 0;
   outputSequence[13,0] := 336;
   outputSequence[13,1] := 298;
   outputSequence[13,2] := 299;
   outputSequence[13,3] := 171;
   outputSequence[13,4] := 65715;
   outputSequence[13,5] := 65739;
   outputSequence[13,6] := 171;
   outputSequence[13,7] := 301;
   outputSequence[13,8] := 134_742_317;
   outputSequence[13,9] := 341;
   outputSequence[13,10..25] := 0;
   outputSequence[14,0] := 336;
   outputSequence[14,1] := 117_440_810;
   outputSequence[14,2] := 299;
   outputSequence[14,3] := 171;
   outputSequence[14,4] := 65715;
   outputSequence[14,5] := 65739;
   outputSequence[14,6] := 171;
   outputSequence[14,7] := 301;
   outputSequence[14,8] := 134_742_317;
   outputSequence[14,9] := 341;
   outputSequence[14,10..25] := 0;
   outputSequence[15,0] := 5408;
   outputSequence[15,1..2] := 4768;
   outputSequence[15,3] := 800;
   outputSequence[15,4] := 11040;
   outputSequence[15,5] := 11424;
   outputSequence[15,6] := 4800;
   outputSequence[15,7] := 37568;
   outputSequence[15,8] := 5440;
   outputSequence[15,9..25] := 0;
   outputSequence[16,0] := 336;
   outputSequence[16,1] := 298;
   outputSequence[16,2] := 299;
   outputSequence[16,3] := 171;
   outputSequence[16,4] := 65715;
   outputSequence[16,5] := 65739;
   outputSequence[16,6] := 171;
   outputSequence[16,7] := 301;
   outputSequence[16,8] := 134_742_317;
   outputSequence[16,9] := 341;
   outputSequence[16,10..25] := 0;
   outputSequence[17,0] := 336;
   outputSequence[17,1] := 298;
   outputSequence[17,2] := 299;
   outputSequence[17,3] := 171;
   outputSequence[17,4] := 65715;
   outputSequence[17,5] := 65739;
   outputSequence[17,6] := 171;
   outputSequence[17,7] := 301;
   outputSequence[17,8] := 134_742_317;
   outputSequence[17,9] := 341;
   outputSequence[17,10..25] := 0;
   outputSequence[18,0] := 336;
   outputSequence[18,1] := 117_440_810;
   outputSequence[18,2] := 117_440_811;
   outputSequence[18,3] := 171;
   outputSequence[18,4] := 65715;
   outputSequence[18,5] := 65739;
   outputSequence[18,6] := 171;
   outputSequence[18,7] := 301;
   outputSequence[18,8] := 940_048_685;
   outputSequence[18,9] := 341;
   outputSequence[18,10..25] := 0;
   outputSequence[19,0] := 336;
   outputSequence[19,1] := 298;
   outputSequence[19,2] := 299;
   outputSequence[19,3] := 171;
   outputSequence[19,4] := 65715;
   outputSequence[19,5] := 65739;
   outputSequence[19,6] := 171;
   outputSequence[19,7] := 301;
   outputSequence[19,8] := 134_742_317;
   outputSequence[19,9] := 341;
   outputSequence[19,10..25] := 0;
   outputSequence[20,0..25] := 0;
   outputSequence[21,0..25] := 0;
   outputSequence[22,0..25] := 0;
   outputSequence[23,0..25] := 0;
   outputSequence[24,0..25] := 0;
   outputSequence[25,0..25] := 0;
   outputSequence[26,0..25] := 0;
   outputSequence[27,0..25] := 0;
   outputSequence[28,0..25] := 0;
   outputSequence[29,0..25] := 0;
   outputSequence[30,0..25] := 0;
   outputSequence[31,0..25] := 0;
   outputSequence[32,0..25] := 0;
   activeOutputsReq[0] := FALSE;
   activeOutputsReq[1] := TRUE;
   activeOutputsReq[2] := FALSE;
   activeOutputsReq[3..4] := TRUE;
   activeOutputsReq[5] := FALSE;
   activeOutputsReq[6] := TRUE;
   activeOutputsReq[7..31] := FALSE;
   maskSequence[0,0..25] := 0;
   maskSequence[1,0..25] := 0;
   maskSequence[2,0..25] := 0;
   maskSequence[3,0..4] := 0;
   maskSequence[3,5..8] := 1024;
   maskSequence[3,9..25] := 0;
   maskSequence[4,0] := 6;
   maskSequence[4,1..2] := 8;
   maskSequence[4,3..4] := 117_440_522;
   maskSequence[4,5] := 117_473_282;
   maskSequence[4,6] := 117_440_522;
   maskSequence[4,7] := -134_283_256;
   maskSequence[4,8] := -135_004_161;
   maskSequence[4,9] := 117_440_512;
   maskSequence[4,10..25] := 0;
   maskSequence[5,0] := -11;
   maskSequence[5,1] := -10;
   maskSequence[5,2] := -11;
   maskSequence[5,3] := -10;
   maskSequence[5,4..25] := 0;
   maskSequence[6,0..25] := 0;
   maskSequence[7,0..25] := 0;
   maskSequence[8,0..25] := 0;
   maskSequence[9,0] := 6;
   maskSequence[9,1..4] := 8;
   maskSequence[9,5] := 32768;
   maskSequence[9,6] := 10;
   maskSequence[9,7] := -134_283_256;
   maskSequence[9,8] := -134_742_017;
   maskSequence[9,9..25] := 0;
   maskSequence[10,0] := 6;
   maskSequence[10,1..4] := 8;
   maskSequence[10,5] := 32768;
   maskSequence[10,6] := 10;
   maskSequence[10,7] := -134_283_256;
   maskSequence[10,8] := -134_742_017;
   maskSequence[10,9..25] := 0;
   maskSequence[11,0] := 6;
   maskSequence[11,1..4] := 8;
   maskSequence[11,5] := 32768;
   maskSequence[11,6] := 10;
   maskSequence[11,7] := -134_283_256;
   maskSequence[11,8] := -134_742_017;
   maskSequence[11,9..25] := 0;
   maskSequence[12,0] := 6;
   maskSequence[12,1..4] := 8;
   maskSequence[12,5] := 32768;
   maskSequence[12,6] := 10;
   maskSequence[12,7] := -134_283_256;
   maskSequence[12,8] := -134_742_017;
   maskSequence[12,9..25] := 0;
   maskSequence[13,0] := 6;
   maskSequence[13,1..4] := 8;
   maskSequence[13,5] := 32768;
   maskSequence[13,6] := 10;
   maskSequence[13,7] := -134_283_256;
   maskSequence[13,8] := -134_742_017;
   maskSequence[13,9..25] := 0;
   maskSequence[14,0] := 6;
   maskSequence[14,1..4] := 8;
   maskSequence[14,5] := 32768;
   maskSequence[14,6] := 10;
   maskSequence[14,7] := -134_283_256;
   maskSequence[14,8] := -134_742_017;
   maskSequence[14,9..25] := 0;
   maskSequence[15,0] := 4096;
   maskSequence[15,1..2] := 0;
   maskSequence[15,3] := 32;
   maskSequence[15,4..25] := 0;
   maskSequence[16,0] := 6;
   maskSequence[16,1..4] := 8;
   maskSequence[16,5] := 32768;
   maskSequence[16,6] := 10;
   maskSequence[16,7] := -134_283_256;
   maskSequence[16,8] := -134_742_017;
   maskSequence[16,9..25] := 0;
   maskSequence[17,0] := 6;
   maskSequence[17,1..4] := 8;
   maskSequence[17,5] := 32768;
   maskSequence[17,6] := 10;
   maskSequence[17,7] := -134_283_256;
   maskSequence[17,8] := -134_742_017;
   maskSequence[17,9..25] := 0;
   maskSequence[18,0] := 117_440_518;
   maskSequence[18,1..2] := 8;
   maskSequence[18,3..4] := 117_440_520;
   maskSequence[18,5] := 117_473_280;
   maskSequence[18,6] := 117_440_522;
   maskSequence[18,7] := -134_283_256;
   maskSequence[18,8] := -940_048_385;
   maskSequence[18,9] := 117_440_512;
   maskSequence[18,10..25] := 0;
   maskSequence[19,0] := 6;
   maskSequence[19,1..4] := 8;
   maskSequence[19,5] := 32768;
   maskSequence[19,6] := 10;
   maskSequence[19,7] := -134_283_256;
   maskSequence[19,8] := -134_742_017;
   maskSequence[19,9..25] := 0;
   maskSequence[20,0..25] := 0;
   maskSequence[21,0..25] := 0;
   maskSequence[22,0..25] := 0;
   maskSequence[23,0..25] := 0;
   maskSequence[24,0..25] := 0;
   maskSequence[25,0..25] := 0;
   maskSequence[26,0..25] := 0;
   maskSequence[27,0..25] := 0;
   maskSequence[28,0..25] := 0;
   maskSequence[29,0..25] := 0;
   maskSequence[30,0..25] := 0;
   maskSequence[31,0..25] := 0;
   maskSequence[32,0..25] := 0;
   activeMask[0..31] := FALSE;
   outputsActive[0] := TRUE;
   outputsActive[1] := FALSE;
   outputsActive[2] := TRUE;
   outputsActive[3] := FALSE;
   outputsActive[4] := TRUE;
   outputsActive[5] := FALSE;
   outputsActive[6] := TRUE;
   outputsActive[7..31] := FALSE;
   text[0] := 'CIL BLOQUEO NIDO IZQ EXT';
   text[1] := 'CIL BLOQUEO NIDO IZQ RET';
   text[2] := 'CIL BLOQUEO NIDO DER EXT';
   text[3] := 'CIL BLOQUEO NIDO DER RET';
   text[4] := 'CIL BLOQUEO TRACK DER EXT';
   text[5] := 'CIL BLOQUEO TRACK DER RET';
   text[6] := 'CIL BLOQUEO TRACK IZQ EXT';
   text[7] := 'CIL BLOQUEO TRACK IZQ RET';
   text[8] := 'ESFUERZO IZQ OK CC15010';
   text[9] := 'ESFUERZO DER OK CC15080';
   text[10] := 'DISTANCIA IZQ INSERCION OK SD14160';
   text[11] := 'DISTANCIA DER INSERCION OK SD14120';
   text[12..15] := 'RESERVA';
   text[16] := 'Prueba motor  izq';
   text[17] := 'Prueba motor derecho';
   text[18..28] := 'Reserva';
   text[29] := 'Imprimir';
   text[30..31] := 'Reserva';
   availableNameManipulate[0] := 'Bloqueo nido izq';
   availableNameManipulate[1] := 'Bloqueo nido der';
   availableNameManipulate[2] := 'Bloqueo track der';
   availableNameManipulate[3] := 'Bloqueo track izq';
   availableNameManipulate[4] := 'Spare 4';
   availableNameManipulate[5] := 'Spare 5';
   availableNameManipulate[6..8] := '';
   status[0] := FALSE;
   status[1] := TRUE;
   status[2] := FALSE;
   status[3] := TRUE;
   status[4] := FALSE;
   status[5] := TRUE;
   status[6] := FALSE;
   status[7] := TRUE;
   status[8..28] := FALSE;
   status[29] := TRUE;
   status[30..63] := FALSE;
   cylinderDirectionA[0..9] := FALSE;
   cylinderDirectionB[0..9] := FALSE;
   cylinderDirectionAActive[0..3] := TRUE;
   cylinderDirectionAActive[4..9] := FALSE;
   cylinderDirectionBActive[0..9] := FALSE;
   cylinderDirectionAStatus[0..9] := FALSE;
   cylinderDirectionBStatus[0..9] := FALSE;
   vent[0..9] := FALSE;
   cylinderStatus[0..9] := 0;
   activateOutput[0] := TRUE;
   activateOutput[1] := FALSE;
   activateOutput[2] := TRUE;
   activateOutput[3] := FALSE;
   activateOutput[4] := TRUE;
   activateOutput[5] := FALSE;
   activateOutput[6] := TRUE;
   activateOutput[7..31] := FALSE;
   timer1.PT := T#0MS;
   timer1.IN := FALSE;
   timer2.PT := T#0MS;
   timer2.IN := FALSE;
   timer3.PT := T#0MS;
   timer3.IN := FALSE;
   timer4.PT := T#0MS;
   timer4.IN := FALSE;
   timer5.PT := T#0MS;
   timer5.IN := FALSE;
   timer6.PT := T#0MS;
   timer6.IN := FALSE;
   timer7.PT := T#0MS;
   timer7.IN := FALSE;
   timer8.PT := T#0MS;
   timer8.IN := FALSE;
   timer9.PT := T#0MS;
   timer9.IN := FALSE;
   timer10.PT := T#0MS;
   timer10.IN := FALSE;
   timer11.PT := T#0MS;
   timer11.IN := FALSE;
   timer12.PT := T#0MS;
   timer12.IN := FALSE;
   timer13.PT := T#0MS;
   timer13.IN := FALSE;
   timer14.PT := T#0MS;
   timer14.IN := FALSE;
   timer15.PT := T#0MS;
   timer15.IN := FALSE;
   timer16.PT := T#0MS;
   timer16.IN := FALSE;
   timer17.PT := T#0MS;
   timer17.IN := FALSE;
   timer18.PT := T#0MS;
   timer18.IN := FALSE;
   timer19.PT := T#0MS;
   timer19.IN := FALSE;
   timer20.PT := T#0MS;
   timer20.IN := FALSE;
   timer21.PT := T#0MS;
   timer21.IN := FALSE;
   timer22.PT := T#0MS;
   timer22.IN := FALSE;
   timer23.PT := T#0MS;
   timer23.IN := FALSE;
   timer24.PT := T#0MS;
   timer24.IN := FALSE;
   timer25.PT := T#0MS;
   timer25.IN := FALSE;
   timer26.PT := T#0MS;
   timer26.IN := FALSE;
   timer27.PT := T#0MS;
   timer27.IN := FALSE;
   timer28.PT := T#0MS;
   timer28.IN := FALSE;
   timer29.PT := T#0MS;
   timer29.IN := FALSE;
   timer30.PT := T#0MS;
   timer30.IN := FALSE;
   timer31.PT := T#0MS;
   timer31.IN := FALSE;
   "timer"[0..31].PT := T#0MS;
   "timer"[0..31].IN := FALSE;
   visibility[0] := FALSE;
   visibility[1..3] := TRUE;
   visibility[4..8] := FALSE;
   energysaverTimer.PT := T#16M;
   energysaverTimer.IN := TRUE;
   scannerOk[0..5] := FALSE;
   scannerLength[0] := 0;
   scannerLength[1] := 3;
   scannerLength[2..3] := 7;
   scannerLength[4..5] := 0;
END_DATA_BLOCK

ORGANIZATION_BLOCK "main"   // OB1, LAD, ProgramCycle
TITLE = "Main Program Sweep (Cycle)"
{ S7_Optimized_Access := 'TRUE' }
VERSION : 0.1
// stored: AutoNumber true, IsIECCheckEnabled false, SetENOAutomatically false
   VAR_INPUT
      Initial_Call : Bool;   // Initial call of this OB
      Remanence : Bool;   // =True, if remanent data are available
   END_VAR
   VAR_TEMP
      BUFFER : String;
   END_VAR
   VAR_TEMP   // added for the SCL form of the ladder/FBD networks
      _w1 : Bool;
      _w2 : Bool;
      _w3 : Bool;
      _w4 : Bool;
      _w5 : Bool;
      _w6 : Bool;
      _w7 : Bool;
      _w8 : Bool;
      _w9 : Bool;
      _w10 : Bool;
   END_VAR
BEGIN

REGION Network 1: SECUENCIA PARA ALARMAR LA MÁQUINA SI SE APAGA A LA MITAD DE UN CICLO DE PRODUCCIÓN
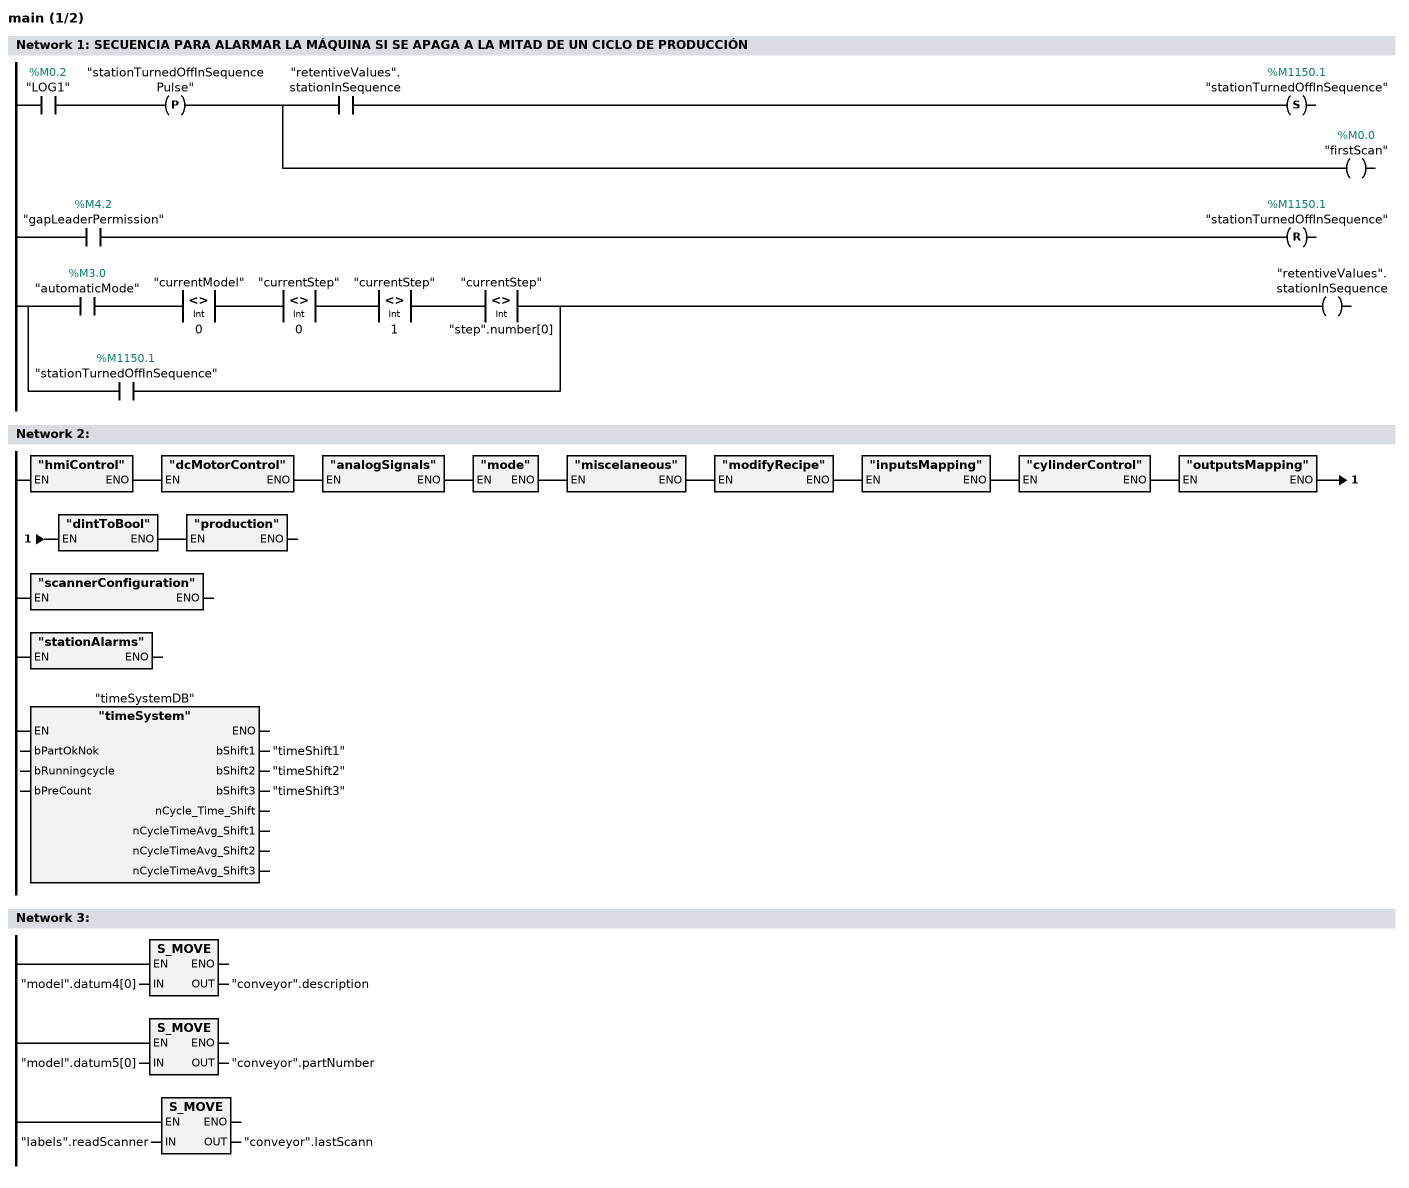
   RUNG wire#powerrail
      Contact( "LOG1" )
      P_Trig( "stationTurnedOffInSequencePulse" )
      wire#w1
      Contact( "retentiveValues".stationInSequence )
      S_Coil( "stationTurnedOffInSequence" )
   END_RUNG
   RUNG wire#w1
      Coil( "firstScan" )
   END_RUNG
   RUNG wire#powerrail
      Contact( "gapLeaderPermission" )
      R_Coil( "stationTurnedOffInSequence" )
   END_RUNG
   RUNG wire#powerrail
      Contact( "automaticMode" )
      { S7_Templates := "SrcType := Int" } NE_Contact(in1 := "currentModel", in2 := 0)
      { S7_Templates := "SrcType := Int" } NE_Contact(in1 := "currentStep", in2 := 0)
      { S7_Templates := "SrcType := Int" } NE_Contact(in1 := "currentStep", in2 := 1)
      { S7_Templates := "SrcType := Int" } NE_Contact(in1 := "currentStep", in2 := "step".number[0])
      wire#w2
      Coil( "retentiveValues".stationInSequence )
   END_RUNG
   RUNG wire#powerrail
      Contact( "stationTurnedOffInSequence" )
   END_RUNG wire#w2
   // the same network as SCL:
   #_w1 := "LOG1" AND NOT "stationTurnedOffInSequencePulse";   // rising edge
   "stationTurnedOffInSequencePulse" := "LOG1";
   IF #_w1 AND "retentiveValues".stationInSequence THEN "stationTurnedOffInSequence" := TRUE; END_IF;
   "firstScan" := #_w1;
   IF "gapLeaderPermission" THEN "stationTurnedOffInSequence" := FALSE; END_IF;
   "retentiveValues".stationInSequence := ("automaticMode" AND ("currentModel" <> 0) AND ("currentStep" <> 0) AND ("currentStep" <> 1) AND ("currentStep" <> "step".number[0])) OR "stationTurnedOffInSequence";
END_REGION

REGION Network 2
   RUNG wire#powerrail
      "hmiControl"()
      "dcMotorControl"()
      "analogSignals"()
      "mode"()
      "miscelaneous"()
      "modifyRecipe"()
      "inputsMapping"()
      "cylinderControl"()
      "outputsMapping"()
      "dintToBool"()
      "production"()
   END_RUNG
   RUNG wire#powerrail
      "scannerConfiguration"()
   END_RUNG
   RUNG wire#powerrail
      "stationAlarms"()
   END_RUNG
   RUNG wire#powerrail
      "timeSystemDB"(bPartOkNok :=, bRunningcycle :=, bPreCount :=, bShift1 => "timeShift1", bShift2 => "timeShift2", bShift3 => "timeShift3", nCycle_Time_Shift =>, nCycleTimeAvg_Shift1 =>, nCycleTimeAvg_Shift2 =>, nCycleTimeAvg_Shift3 =>)
   END_RUNG
   // the same network as SCL:
   "hmiControl"(ENO => #_w1);
   "dcMotorControl"(EN := #_w1, ENO => #_w2);
   "analogSignals"(EN := #_w2, ENO => #_w3);
   "mode"(EN := #_w3, ENO => #_w4);
   "miscelaneous"(EN := #_w4, ENO => #_w5);
   "modifyRecipe"(EN := #_w5, ENO => #_w6);
   "inputsMapping"(EN := #_w6, ENO => #_w7);
   "cylinderControl"(EN := #_w7, ENO => #_w8);
   "outputsMapping"(EN := #_w8, ENO => #_w9);
   "dintToBool"(EN := #_w9, ENO => #_w10);
   IF #_w10 THEN "production"(); END_IF;
   "scannerConfiguration"();
   "stationAlarms"();
   "timeSystemDB"(bShift1 => "timeShift1", bShift2 => "timeShift2", bShift3 => "timeShift3");   // "timeSystem"
END_REGION

REGION Network 3
   RUNG wire#powerrail
      S_Move(in := "model".datum4[0], out => "conveyor".description)
   END_RUNG
   RUNG wire#powerrail
      S_Move(in := "model".datum5[0], out => "conveyor".partNumber)
   END_RUNG
   RUNG wire#powerrail
      S_Move(in := "labels".readScanner, out => "conveyor".lastScann)
   END_RUNG
   // the same network as SCL:
   "conveyor".description := "model".datum4[0];
   "conveyor".partNumber := "model".datum5[0];
   "conveyor".lastScann := "labels".readScanner;
END_REGION

REGION Network 4: Permissions
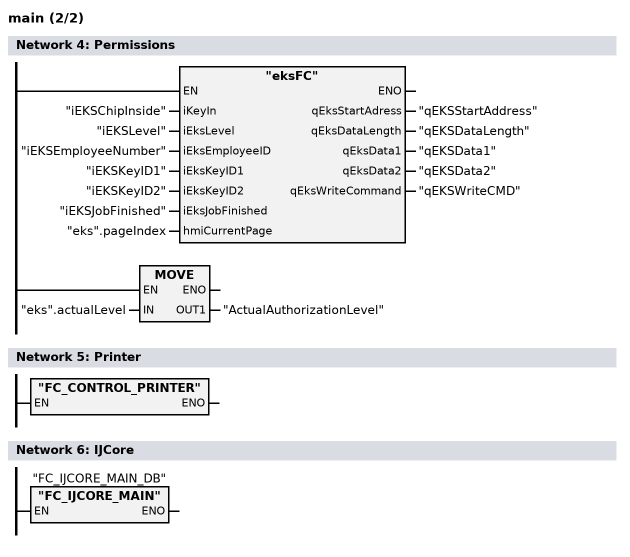
   RUNG wire#powerrail
      "eksFC"(iKeyIn := "iEKSChipInside", iEksLevel := "iEKSLevel", iEksEmployeeID := "iEKSEmployeeNumber", iEksKeyID1 := "iEKSKeyID1", iEksKeyID2 := "iEKSKeyID2", iEksJobFinished := "iEKSJobFinished", hmiCurrentPage := "eks".pageIndex, qEksStartAdress => "qEKSStartAddress", qEksDataLength => "qEKSDataLength", qEksData1 => "qEKSData1", qEksData2 => "qEKSData2", qEksWriteCommand => "qEKSWriteCMD")
   END_RUNG
   RUNG wire#powerrail
      Move(in := "eks".actualLevel, out1 => "ActualAuthorizationLevel")
   END_RUNG
   // the same network as SCL:
   "eksFC"(iKeyIn := "iEKSChipInside",
           iEksLevel := "iEKSLevel",
           iEksEmployeeID := "iEKSEmployeeNumber",
           iEksKeyID1 := "iEKSKeyID1",
           iEksKeyID2 := "iEKSKeyID2",
           iEksJobFinished := "iEKSJobFinished",
           hmiCurrentPage := "eks".pageIndex,
           qEksStartAdress => "qEKSStartAddress",
           qEksDataLength => "qEKSDataLength",
           qEksData1 => "qEKSData1",
           qEksData2 => "qEKSData2",
           qEksWriteCommand => "qEKSWriteCMD");
   "ActualAuthorizationLevel" := "eks".actualLevel;
END_REGION

REGION Network 5: Printer
   RUNG wire#powerrail
      "FC_CONTROL_PRINTER"()
   END_RUNG
   // the same network as SCL:
   "FC_CONTROL_PRINTER"();
END_REGION

REGION Network 6: IJCore
   RUNG wire#powerrail
      "FC_IJCORE_MAIN_DB"()
   END_RUNG
   // the same network as SCL:
   "FC_IJCORE_MAIN_DB"();   // "FC_IJCORE_MAIN"
END_REGION
END_ORGANIZATION_BLOCK

FUNCTION "hmiControl" : Void   // FC3, LAD
{ S7_Optimized_Access := 'TRUE' }
VERSION : 0.1
// stored: AutoNumber true, IsIECCheckEnabled false, SetENOAutomatically false, UDAEnableTagReadback false
   VAR_TEMP   // added for the SCL form of the ladder/FBD networks
      _w1 : Bool;
      _w2 : Bool;
      _w3 : Bool;
      _w4 : Bool;
      _w5 : Bool;
      _w6 : Bool;
      _w7 : Bool;
      _w8 : Bool;
      _w9 : Bool;
      _w10 : Bool;
      _w11 : Bool;
      _w12 : Bool;
      _w13 : Bool;
      _w14 : Bool;
      _w15 : Bool;
      _w16 : Bool;
      _w17 : Bool;
      _w18 : Bool;
      _w19 : Bool;
      _w20 : Bool;
      _w21 : Bool;
      _w22 : Bool;
      _w23 : Bool;
      _w24 : Bool;
      _w25 : Bool;
      _w26 : Bool;
      _w27 : Bool;
      _w28 : Bool;
      _w29 : Bool;
      _w30 : Bool;
      _w31 : Bool;
      _w32 : Bool;
   END_VAR
BEGIN

REGION Network 1: MODEL VISUALIZATION: IF EVERY MODEL HAS A NAME RECORDED, ITS VISUALIZATION IS ACTIVATED
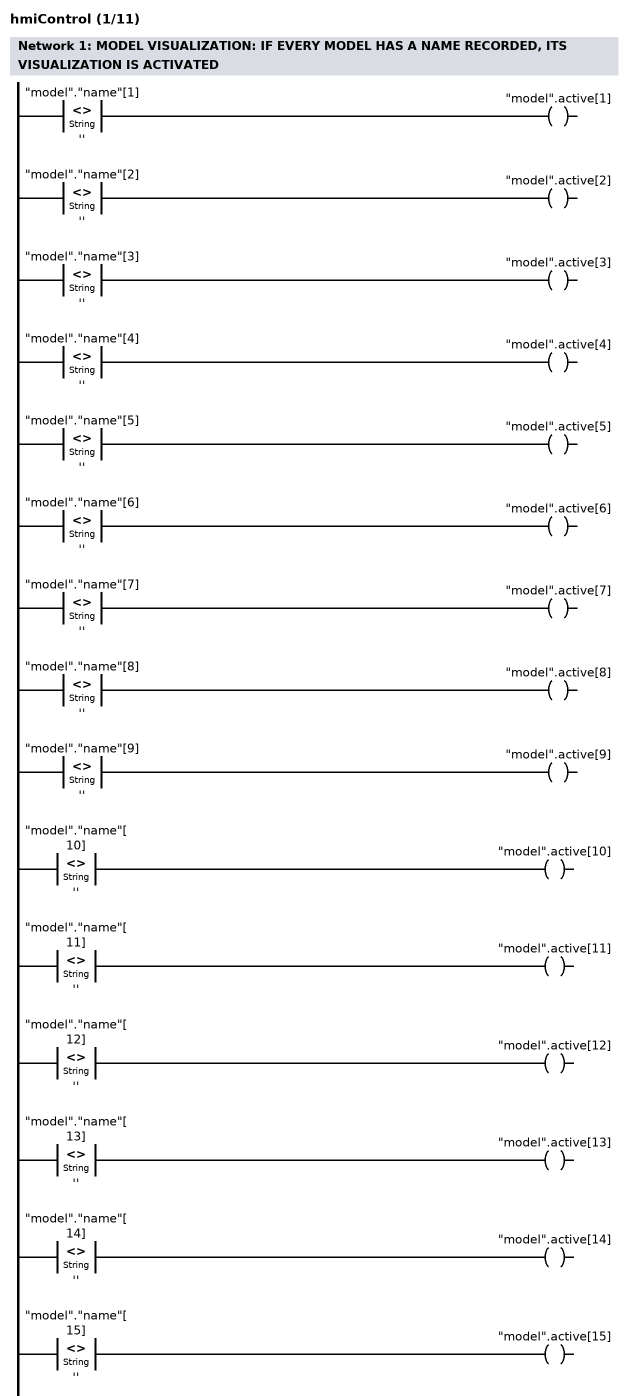
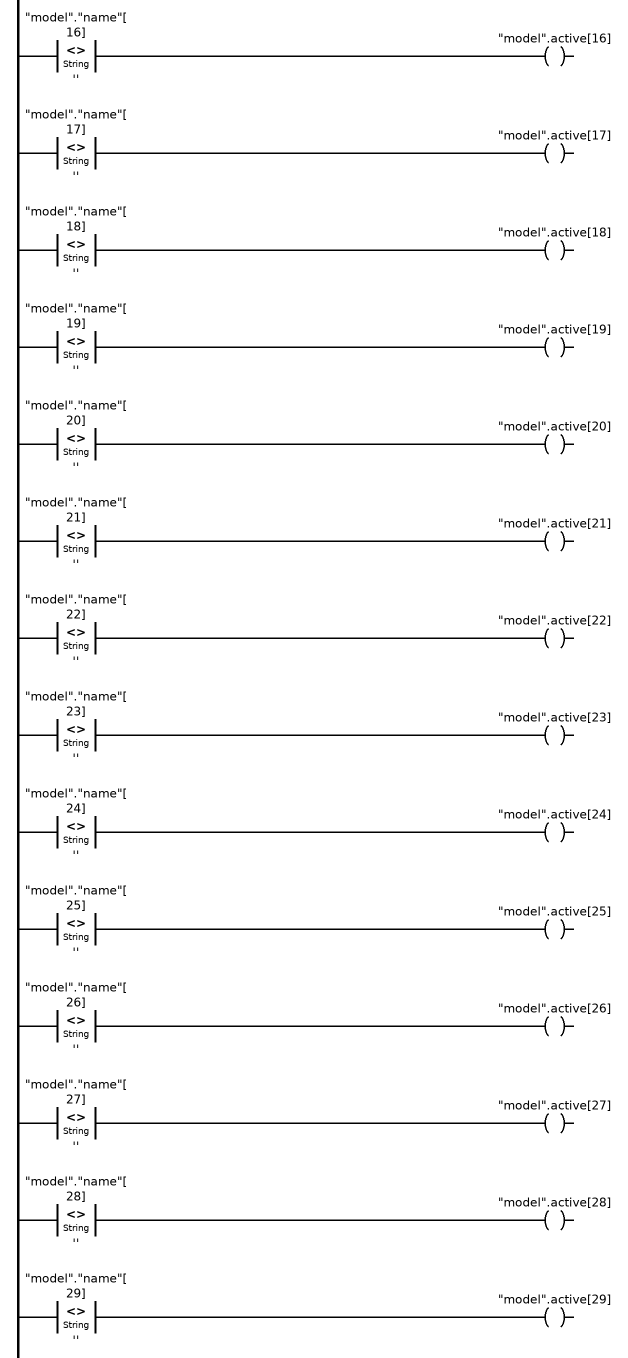
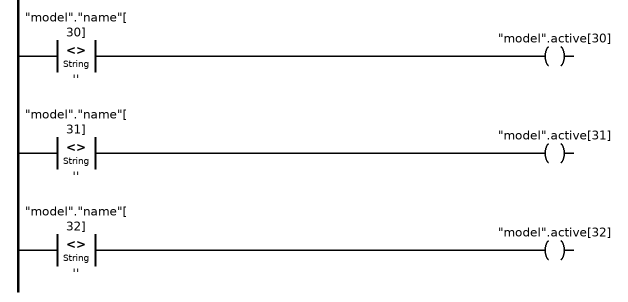
   RUNG wire#powerrail
      { S7_Templates := "SrcType := String" } NE_Contact(in1 := "model"."name"[1], in2 := '')
      Coil( "model".active[1] )
   END_RUNG
   RUNG wire#powerrail
      { S7_Templates := "SrcType := String" } NE_Contact(in1 := "model"."name"[2], in2 := '')
      Coil( "model".active[2] )
   END_RUNG
   RUNG wire#powerrail
      { S7_Templates := "SrcType := String" } NE_Contact(in1 := "model"."name"[3], in2 := '')
      Coil( "model".active[3] )
   END_RUNG
   RUNG wire#powerrail
      { S7_Templates := "SrcType := String" } NE_Contact(in1 := "model"."name"[4], in2 := '')
      Coil( "model".active[4] )
   END_RUNG
   RUNG wire#powerrail
      { S7_Templates := "SrcType := String" } NE_Contact(in1 := "model"."name"[5], in2 := '')
      Coil( "model".active[5] )
   END_RUNG
   RUNG wire#powerrail
      { S7_Templates := "SrcType := String" } NE_Contact(in1 := "model"."name"[6], in2 := '')
      Coil( "model".active[6] )
   END_RUNG
   RUNG wire#powerrail
      { S7_Templates := "SrcType := String" } NE_Contact(in1 := "model"."name"[7], in2 := '')
      Coil( "model".active[7] )
   END_RUNG
   RUNG wire#powerrail
      { S7_Templates := "SrcType := String" } NE_Contact(in1 := "model"."name"[8], in2 := '')
      Coil( "model".active[8] )
   END_RUNG
   RUNG wire#powerrail
      { S7_Templates := "SrcType := String" } NE_Contact(in1 := "model"."name"[9], in2 := '')
      Coil( "model".active[9] )
   END_RUNG
   RUNG wire#powerrail
      { S7_Templates := "SrcType := String" } NE_Contact(in1 := "model"."name"[10], in2 := '')
      Coil( "model".active[10] )
   END_RUNG
   RUNG wire#powerrail
      { S7_Templates := "SrcType := String" } NE_Contact(in1 := "model"."name"[11], in2 := '')
      Coil( "model".active[11] )
   END_RUNG
   RUNG wire#powerrail
      { S7_Templates := "SrcType := String" } NE_Contact(in1 := "model"."name"[12], in2 := '')
      Coil( "model".active[12] )
   END_RUNG
   RUNG wire#powerrail
      { S7_Templates := "SrcType := String" } NE_Contact(in1 := "model"."name"[13], in2 := '')
      Coil( "model".active[13] )
   END_RUNG
   RUNG wire#powerrail
      { S7_Templates := "SrcType := String" } NE_Contact(in1 := "model"."name"[14], in2 := '')
      Coil( "model".active[14] )
   END_RUNG
   RUNG wire#powerrail
      { S7_Templates := "SrcType := String" } NE_Contact(in1 := "model"."name"[15], in2 := '')
      Coil( "model".active[15] )
   END_RUNG
   RUNG wire#powerrail
      { S7_Templates := "SrcType := String" } NE_Contact(in1 := "model"."name"[16], in2 := '')
      Coil( "model".active[16] )
   END_RUNG
   RUNG wire#powerrail
      { S7_Templates := "SrcType := String" } NE_Contact(in1 := "model"."name"[17], in2 := '')
      Coil( "model".active[17] )
   END_RUNG
   RUNG wire#powerrail
      { S7_Templates := "SrcType := String" } NE_Contact(in1 := "model"."name"[18], in2 := '')
      Coil( "model".active[18] )
   END_RUNG
   RUNG wire#powerrail
      { S7_Templates := "SrcType := String" } NE_Contact(in1 := "model"."name"[19], in2 := '')
      Coil( "model".active[19] )
   END_RUNG
   RUNG wire#powerrail
      { S7_Templates := "SrcType := String" } NE_Contact(in1 := "model"."name"[20], in2 := '')
      Coil( "model".active[20] )
   END_RUNG
   RUNG wire#powerrail
      { S7_Templates := "SrcType := String" } NE_Contact(in1 := "model"."name"[21], in2 := '')
      Coil( "model".active[21] )
   END_RUNG
   RUNG wire#powerrail
      { S7_Templates := "SrcType := String" } NE_Contact(in1 := "model"."name"[22], in2 := '')
      Coil( "model".active[22] )
   END_RUNG
   RUNG wire#powerrail
      { S7_Templates := "SrcType := String" } NE_Contact(in1 := "model"."name"[23], in2 := '')
      Coil( "model".active[23] )
   END_RUNG
   RUNG wire#powerrail
      { S7_Templates := "SrcType := String" } NE_Contact(in1 := "model"."name"[24], in2 := '')
      Coil( "model".active[24] )
   END_RUNG
   RUNG wire#powerrail
      { S7_Templates := "SrcType := String" } NE_Contact(in1 := "model"."name"[25], in2 := '')
      Coil( "model".active[25] )
   END_RUNG
   RUNG wire#powerrail
      { S7_Templates := "SrcType := String" } NE_Contact(in1 := "model"."name"[26], in2 := '')
      Coil( "model".active[26] )
   END_RUNG
   RUNG wire#powerrail
      { S7_Templates := "SrcType := String" } NE_Contact(in1 := "model"."name"[27], in2 := '')
      Coil( "model".active[27] )
   END_RUNG
   RUNG wire#powerrail
      { S7_Templates := "SrcType := String" } NE_Contact(in1 := "model"."name"[28], in2 := '')
      Coil( "model".active[28] )
   END_RUNG
   RUNG wire#powerrail
      { S7_Templates := "SrcType := String" } NE_Contact(in1 := "model"."name"[29], in2 := '')
      Coil( "model".active[29] )
   END_RUNG
   RUNG wire#powerrail
      { S7_Templates := "SrcType := String" } NE_Contact(in1 := "model"."name"[30], in2 := '')
      Coil( "model".active[30] )
   END_RUNG
   RUNG wire#powerrail
      { S7_Templates := "SrcType := String" } NE_Contact(in1 := "model"."name"[31], in2 := '')
      Coil( "model".active[31] )
   END_RUNG
   RUNG wire#powerrail
      { S7_Templates := "SrcType := String" } NE_Contact(in1 := "model"."name"[32], in2 := '')
      Coil( "model".active[32] )
   END_RUNG
   // the same network as SCL:
   "model".active[1] := "model"."name"[1] <> '';
   "model".active[2] := "model"."name"[2] <> '';
   "model".active[3] := "model"."name"[3] <> '';
   "model".active[4] := "model"."name"[4] <> '';
   "model".active[5] := "model"."name"[5] <> '';
   "model".active[6] := "model"."name"[6] <> '';
   "model".active[7] := "model"."name"[7] <> '';
   "model".active[8] := "model"."name"[8] <> '';
   "model".active[9] := "model"."name"[9] <> '';
   "model".active[10] := "model"."name"[10] <> '';
   "model".active[11] := "model"."name"[11] <> '';
   "model".active[12] := "model"."name"[12] <> '';
   "model".active[13] := "model"."name"[13] <> '';
   "model".active[14] := "model"."name"[14] <> '';
   "model".active[15] := "model"."name"[15] <> '';
   "model".active[16] := "model"."name"[16] <> '';
   "model".active[17] := "model"."name"[17] <> '';
   "model".active[18] := "model"."name"[18] <> '';
   "model".active[19] := "model"."name"[19] <> '';
   "model".active[20] := "model"."name"[20] <> '';
   "model".active[21] := "model"."name"[21] <> '';
   "model".active[22] := "model"."name"[22] <> '';
   "model".active[23] := "model"."name"[23] <> '';
   "model".active[24] := "model"."name"[24] <> '';
   "model".active[25] := "model"."name"[25] <> '';
   "model".active[26] := "model"."name"[26] <> '';
   "model".active[27] := "model"."name"[27] <> '';
   "model".active[28] := "model"."name"[28] <> '';
   "model".active[29] := "model"."name"[29] <> '';
   "model".active[30] := "model"."name"[30] <> '';
   "model".active[31] := "model"."name"[31] <> '';
   "model".active[32] := "model"."name"[32] <> '';
END_REGION

